# B&R Automation Studio project NAEUL004C00R13L518F00 (part 52)

#### Act_Main.st - Do Not Change!!!
```iecst
(** 2020-03-16 **)
ACTION Act_Main:

	IF bModuleNotOK = FALSE THEN
		CASE eStat OF

			LifterActIdle:
				IF eStatus <> Idle THEN	//Reset Data
					//Private
					fbStop(bEn := FALSE);
					fbRstAxisErr(bEn := FALSE);
					fbJog(bEn := FALSE);
					fbMovRel(bEn := FALSE);
					fbMovAbs(bEn := FALSE);
					fbHoming(bEn := FALSE);
					fbPwrOff(bEn := FALSE);
					fbPwrOn(bEn := FALSE);
					fbFullHm(bEn := FALSE);
					fbFullMovAbs(bEn := FALSE);
					fbFullMovRel(bEn := FALSE);
					fbSDOWrite(bEn := FALSE);
					fbTm(IN := FALSE);
					usiStep	:= 0;
					usiCount			:= 0;
					bNotInterruptible	:= FALSE;

					sStatTxt	:= a_sStatText[eStat];

				END_IF

				eStatus	:= Idle;

				IF EDGENEG(p_bManual) THEN
					fMotionCANRstCtrlWord(ADR(tyParamOutDriver));
				END_IF

			LifterActGoAPos:
				IF (eStatus = Idle OR eStatus = Busy) THEN

					eStatus	:= Busy;

					sStatTxt	:= a_sStatText[eStat];

					bNotInterruptible	:= TRUE;

					CASE usiStep OF
						0:	//Wait For Motion Parameter Update
							p_diMovePosInUM	:= p_diAPos;
							usiStep	:= 1;

						1:	//Check Position Difference
							IF tyParamOut.bPosDiff = TRUE THEN
								usiStep	:= 2;
							ELSE
								eStatus	:= Done;
							END_IF

						2:	//Move
							fbFullMovAbs.tyParamInDriver					:= tyParamInDriver;
							fbFullMovAbs.tyParamInMove.diPosInUM			:= p_diMovePosInUM;
							fbFullMovAbs.tyParamInMove.diDistInUM			:= p_diMoveDistInUM;
							fbFullMovAbs.tyParamInMove.diVelInUMPS			:= p_diMoveVelInUMPS;
							fbFullMovAbs.tyParamInMove.diAcc				:= p_diMoveAcc;
							fbFullMovAbs.tyParamInMove.diDec				:= p_diMoveDec;
							fbFullMovAbs.tyParamOut							:= tyParamOut;
							fbFullMovAbs(bEn := TRUE);

							IF fbFullMovAbs.udiStatus = 0 THEN
								eStatus	:= Done;
							ELSIF fbFullMovAbs.udiStatus < 65534 THEN
								eStatus		:= Error;

								IF fbFullMovAbs.udiStatus = 1401 THEN
									udiStatus	:= 10002;	//Power On Time Out While Going A Position
								ELSIF fbFullMovAbs.udiStatus = 1402 THEN
									udiStatus	:= 10003;	//Homing Time Out While Going A Position
								ELSIF fbFullMovAbs.udiStatus = 1403 THEN
									udiStatus	:= 10004;	//Move Absolute Time Out While Going A Position
								ELSIF fbFullMovAbs.udiStatus = 1405 THEN
									udiStatus	:= 10005;	//Stop Motion Time Out While Going A Position
								ELSIF fbFullMovAbs.udiStatus = 1408 THEN
									udiStatus	:= 10006;	//Axis Error Reset Failed While Going A Position
								ELSIF fbFullMovAbs.udiStatus = 1409 THEN
									udiStatus	:= 10007;	//Axis Error Occur In Move Absolute While Going A Position
								ELSIF fbFullMovAbs.udiStatus = 1411 THEN
									udiStatus	:= 10008;	//Axis Error Occur In Homing While Going A Position
								ELSIF fbFullMovAbs.udiStatus = 1412 THEN
									udiStatus	:= 10009;	//Homing Done But Home Flag Is Not Activated While Going A Position
								ELSIF fbFullMovAbs.udiStatus = 1413 THEN
									udiStatus	:= 10010;	//Forward Limit Activated In Homing While Going A Position
								ELSIF fbFullMovAbs.udiStatus = 1414 THEN
									udiStatus	:= 10011;	//Reverse Limit Activated In Homing While Going A Position
								ELSIF fbFullMovAbs.udiStatus = 1415 THEN
									udiStatus	:= 10012;	//Forward Limit Activated In Move Absolute While Going A Position
								ELSIF fbFullMovAbs.udiStatus = 1416 THEN
									udiStatus	:= 10013;	//Reverse Limit Activated In Move Absolute While Going A Position
								ELSE
									udiStatus	:= fbFullMovAbs.udiStatus;
								END_IF
							END_IF

					END_CASE

				END_IF

			LifterActGoBPos:
				IF (eStatus = Idle OR eStatus = Busy) THEN

					eStatus	:= Busy;

					sStatTxt	:= a_sStatText[eStat];

					bNotInterruptible	:= TRUE;

					CASE usiStep OF
						0:	//Wait For Motion Parameter Update
							p_diMovePosInUM	:= p_diBPos;
							usiStep	:= 1;

						1:	//Check Position Difference
							IF tyParamOut.bPosDiff = TRUE THEN
								usiStep	:= 2;
							ELSE
								eStatus	:= Done;
							END_IF

						2:	//Move
							fbFullMovAbs.tyParamInDriver					:= tyParamInDriver;
							fbFullMovAbs.tyParamInMove.diPosInUM			:= p_diMovePosInUM;
							fbFullMovAbs.tyParamInMove.diDistInUM			:= p_diMoveDistInUM;
							fbFullMovAbs.tyParamInMove.diVelInUMPS			:= p_diMoveVelInUMPS;
							fbFullMovAbs.tyParamInMove.diAcc				:= p_diMoveAcc;
							fbFullMovAbs.tyParamInMove.diDec				:= p_diMoveDec;
							fbFullMovAbs.tyParamOut							:= tyParamOut;
							fbFullMovAbs(bEn := TRUE);

							IF fbFullMovAbs.udiStatus = 0 THEN
								eStatus	:= Done;
							ELSIF fbFullMovAbs.udiStatus < 65534 THEN
								eStatus		:= Error;

								IF fbFullMovAbs.udiStatus = 1401 THEN
									udiStatus	:= 10029;	//Power On Time Out While Going B Position
								ELSIF fbFullMovAbs.udiStatus = 1402 THEN
									udiStatus	:= 10030;	//Homing Time Out While Going B Position
								ELSIF fbFullMovAbs.udiStatus = 1403 THEN
									udiStatus	:= 10031;	//Move Absolute Time Out While Going B Position
								ELSIF fbFullMovAbs.udiStatus = 1405 THEN
									udiStatus	:= 10032;	//Stop Motion Time Out While Going B Position
								ELSIF fbFullMovAbs.udiStatus = 1408 THEN
									udiStatus	:= 10033;	//Axis Error Reset Failed While Going B Position
								ELSIF fbFullMovAbs.udiStatus = 1409 THEN
									udiStatus	:= 10034;	//Axis Error Occur In Move Absolute While Going B Position
								ELSIF fbFullMovAbs.udiStatus = 1411 THEN
									udiStatus	:= 10035;	//Axis Error Occur In Homing While Going B Position
								ELSIF fbFullMovAbs.udiStatus = 1412 THEN
									udiStatus	:= 10036;	//Homing Done But Home Flag Is Not Activated While Going B Position
								ELSIF fbFullMovAbs.udiStatus = 1413 THEN
									udiStatus	:= 10037;	//Forward Limit Activated In Homing While Going B Position
								ELSIF fbFullMovAbs.udiStatus = 1414 THEN
									udiStatus	:= 10038;	//Reverse Limit Activated In Homing While Going B Position
								ELSIF fbFullMovAbs.udiStatus = 1415 THEN
									udiStatus	:= 10039;	//Forward Limit Activated In Move Absolute While Going B Position
								ELSIF fbFullMovAbs.udiStatus = 1416 THEN
									udiStatus	:= 10040;	//Reverse Limit Activated In Move Absolute While Going B Position
								ELSE
									udiStatus	:= fbFullMovAbs.udiStatus;
								END_IF
							END_IF

					END_CASE

				END_IF

			LifterActGoCPos:
				IF (eStatus = Idle OR eStatus = Busy) THEN

					eStatus	:= Busy;

					sStatTxt	:= a_sStatText[eStat];

					bNotInterruptible	:= TRUE;

					CASE usiStep OF
						0:	//Wait For Motion Parameter Update
							p_diMovePosInUM	:= p_diCPos;
							usiStep	:= 1;

						1:	//Check Position Difference
							IF tyParamOut.bPosDiff = TRUE THEN
								usiStep	:= 2;
							ELSE
								eStatus	:= Done;
							END_IF

						2:	//Move
							fbFullMovAbs.tyParamInDriver					:= tyParamInDriver;
							fbFullMovAbs.tyParamInMove.diPosInUM			:= p_diMovePosInUM;
							fbFullMovAbs.tyParamInMove.diDistInUM			:= p_diMoveDistInUM;
							fbFullMovAbs.tyParamInMove.diVelInUMPS			:= p_diMoveVelInUMPS;
							fbFullMovAbs.tyParamInMove.diAcc				:= p_diMoveAcc;
							fbFullMovAbs.tyParamInMove.diDec				:= p_diMoveDec;
							fbFullMovAbs.tyParamOut							:= tyParamOut;
							fbFullMovAbs(bEn := TRUE);

							IF fbFullMovAbs.udiStatus = 0 THEN
								eStatus	:= Done;
							ELSIF fbFullMovAbs.udiStatus < 65534 THEN
								eStatus		:= Error;

								IF fbFullMovAbs.udiStatus = 1401 THEN
									udiStatus	:= 10078;	//Power On Time Out While Going C Position
								ELSIF fbFullMovAbs.udiStatus = 1402 THEN
									udiStatus	:= 10079;	//Homing Time Out While Going C Position
								ELSIF fbFullMovAbs.udiStatus = 1403 THEN
									udiStatus	:= 10080;	//Move Absolute Time Out While Going C Position
								ELSIF fbFullMovAbs.udiStatus = 1405 THEN
									udiStatus	:= 10081;	//Stop Motion Time Out While Going C Position
								ELSIF fbFullMovAbs.udiStatus = 1408 THEN
									udiStatus	:= 10082;	//Axis Error Reset Failed While Going C Position
								ELSIF fbFullMovAbs.udiStatus = 1409 THEN
									udiStatus	:= 10083;	//Axis Error Occur In Move Absolute While Going C Position
								ELSIF fbFullMovAbs.udiStatus = 1411 THEN
									udiStatus	:= 10084;	//Axis Error Occur In Homing While Going C Position
								ELSIF fbFullMovAbs.udiStatus = 1412 THEN
									udiStatus	:= 10085;	//Homing Done But Home Flag Is Not Activated While Going C Position
								ELSIF fbFullMovAbs.udiStatus = 1413 THEN
									udiStatus	:= 10086;	//Forward Limit Activated In Homing While Going C Position
								ELSIF fbFullMovAbs.udiStatus = 1414 THEN
									udiStatus	:= 10087;	//Reverse Limit Activated In Homing While Going C Position
								ELSIF fbFullMovAbs.udiStatus = 1415 THEN
									udiStatus	:= 10088;	//Forward Limit Activated In Move Absolute While Going C Position
								ELSIF fbFullMovAbs.udiStatus = 1416 THEN
									udiStatus	:= 10089;	//Reverse Limit Activated In Move Absolute While Going C Position
								ELSE
									udiStatus	:= fbFullMovAbs.udiStatus;
								END_IF
							END_IF

					END_CASE

				END_IF

			LifterActGoDPos:
				IF (eStatus = Idle OR eStatus = Busy) THEN

					eStatus	:= Busy;

					sStatTxt	:= a_sStatText[eStat];

					bNotInterruptible	:= TRUE;

					CASE usiStep OF
						0:	//Wait For Motion Parameter Update
							p_diMovePosInUM	:= p_diDPos;
							usiStep	:= 1;

						1:	//Check Position Difference
							IF tyParamOut.bPosDiff = TRUE THEN
								usiStep	:= 2;
							ELSE
								eStatus	:= Done;
							END_IF

						2:	//Move
							fbFullMovAbs.tyParamInDriver					:= tyParamInDriver;
							fbFullMovAbs.tyParamInMove.diPosInUM			:= p_diMovePosInUM;
							fbFullMovAbs.tyParamInMove.diDistInUM			:= p_diMoveDistInUM;
							fbFullMovAbs.tyParamInMove.diVelInUMPS			:= p_diMoveVelInUMPS;
							fbFullMovAbs.tyParamInMove.diAcc				:= p_diMoveAcc;
							fbFullMovAbs.tyParamInMove.diDec				:= p_diMoveDec;
							fbFullMovAbs.tyParamOut							:= tyParamOut;
							fbFullMovAbs(bEn := TRUE);

							IF fbFullMovAbs.udiStatus = 0 THEN
								eStatus	:= Done;
							ELSIF fbFullMovAbs.udiStatus < 65534 THEN
								eStatus		:= Error;

								IF fbFullMovAbs.udiStatus = 1401 THEN
									udiStatus	:= 10090;	//Power On Time Out While Going D Position
								ELSIF fbFullMovAbs.udiStatus = 1402 THEN
									udiStatus	:= 10091;	//Homing Time Out While Going D Position
								ELSIF fbFullMovAbs.udiStatus = 1403 THEN
									udiStatus	:= 10092;	//Move Absolute Time Out While Going D Position
								ELSIF fbFullMovAbs.udiStatus = 1405 THEN
									udiStatus	:= 10093;	//Stop Motion Time Out While Going D Position
								ELSIF fbFullMovAbs.udiStatus = 1408 THEN
									udiStatus	:= 10094;	//Axis Error Reset Failed While Going D Position
								ELSIF fbFullMovAbs.udiStatus = 1409 THEN
									udiStatus	:= 10095;	//Axis Error Occur In Move Absolute While Going D Position
								ELSIF fbFullMovAbs.udiStatus = 1411 THEN
									udiStatus	:= 10096;	//Axis Error Occur In Homing While Going D Position
								ELSIF fbFullMovAbs.udiStatus = 1412 THEN
									udiStatus	:= 10097;	//Homing Done But Home Flag Is Not Activated While Going D Position
								ELSIF fbFullMovAbs.udiStatus = 1413 THEN
									udiStatus	:= 10098;	//Forward Limit Activated In Homing While Going D Position
								ELSIF fbFullMovAbs.udiStatus = 1414 THEN
									udiStatus	:= 10099;	//Reverse Limit Activated In Homing While Going D Position
								ELSIF fbFullMovAbs.udiStatus = 1415 THEN
									udiStatus	:= 10100;	//Forward Limit Activated In Move Absolute While Going D Position
								ELSIF fbFullMovAbs.udiStatus = 1416 THEN
									udiStatus	:= 10101;	//Reverse Limit Activated In Move Absolute While Going D Position
								ELSE
									udiStatus	:= fbFullMovAbs.udiStatus;
								END_IF
							END_IF

					END_CASE

				END_IF

			LifterActGoEPos:
				IF (eStatus = Idle OR eStatus = Busy) THEN

					eStatus	:= Busy;

					sStatTxt	:= a_sStatText[eStat];

					bNotInterruptible	:= TRUE;

					CASE usiStep OF
						0:	//Wait For Motion Parameter Update
							p_diMovePosInUM	:= p_diEPos;
							usiStep	:= 1;

						1:	//Check Position Difference
							IF tyParamOut.bPosDiff = TRUE THEN
								usiStep	:= 2;
							ELSE
								eStatus	:= Done;
							END_IF

						2:	//Move
							fbFullMovAbs.tyParamInDriver					:= tyParamInDriver;
							fbFullMovAbs.tyParamInMove.diPosInUM			:= p_diMovePosInUM;
							fbFullMovAbs.tyParamInMove.diDistInUM			:= p_diMoveDistInUM;
							fbFullMovAbs.tyParamInMove.diVelInUMPS			:= p_diMoveVelInUMPS;
							fbFullMovAbs.tyParamInMove.diAcc				:= p_diMoveAcc;
							fbFullMovAbs.tyParamInMove.diDec				:= p_diMoveDec;
							fbFullMovAbs.tyParamOut							:= tyParamOut;
							fbFullMovAbs(bEn := TRUE);

							IF fbFullMovAbs.udiStatus = 0 THEN
								eStatus	:= Done;
							ELSIF fbFullMovAbs.udiStatus < 65534 THEN
								eStatus		:= Error;

								IF fbFullMovAbs.udiStatus = 1401 THEN
									udiStatus	:= 10102;	//Power On Time Out While Going E Position
								ELSIF fbFullMovAbs.udiStatus = 1402 THEN
									udiStatus	:= 10103;	//Homing Time Out While Going E Position
								ELSIF fbFullMovAbs.udiStatus = 1403 THEN
									udiStatus	:= 10104;	//Move Absolute Time Out While Going E Position
								ELSIF fbFullMovAbs.udiStatus = 1405 THEN
									udiStatus	:= 10105;	//Stop Motion Time Out While Going E Position
								ELSIF fbFullMovAbs.udiStatus = 1408 THEN
									udiStatus	:= 10106;	//Axis Error Reset Failed While Going E Position
								ELSIF fbFullMovAbs.udiStatus = 1409 THEN
									udiStatus	:= 10107;	//Axis Error Occur In Move Absolute While Going E Position
								ELSIF fbFullMovAbs.udiStatus = 1411 THEN
									udiStatus	:= 10108;	//Axis Error Occur In Homing While Going E Position
								ELSIF fbFullMovAbs.udiStatus = 1412 THEN
									udiStatus	:= 10109;	//Homing Done But Home Flag Is Not Activated While Going E Position
								ELSIF fbFullMovAbs.udiStatus = 1413 THEN
									udiStatus	:= 10110;	//Forward Limit Activated In Homing While Going E Position
								ELSIF fbFullMovAbs.udiStatus = 1414 THEN
									udiStatus	:= 10111;	//Reverse Limit Activated In Homing While Going E Position
								ELSIF fbFullMovAbs.udiStatus = 1415 THEN
									udiStatus	:= 10112;	//Forward Limit Activated In Move Absolute While Going E Position
								ELSIF fbFullMovAbs.udiStatus = 1416 THEN
									udiStatus	:= 10113;	//Reverse Limit Activated In Move Absolute While Going E Position
								ELSE
									udiStatus	:= fbFullMovAbs.udiStatus;
								END_IF
							END_IF

					END_CASE

				END_IF

			LifterActGoFPos:
				IF (eStatus = Idle OR eStatus = Busy) THEN

					eStatus	:= Busy;

					sStatTxt	:= a_sStatText[eStat];

					bNotInterruptible	:= TRUE;

					CASE usiStep OF
						0:	//Wait For Motion Parameter Update
							p_diMovePosInUM	:= p_diFPos;
							usiStep	:= 1;

						1:	//Check Position Difference
							IF tyParamOut.bPosDiff = TRUE THEN
								usiStep	:= 2;
							ELSE
								eStatus	:= Done;
							END_IF

						2:	//Move
							fbFullMovAbs.tyParamInDriver					:= tyParamInDriver;
							fbFullMovAbs.tyParamInMove.diPosInUM			:= p_diMovePosInUM;
							fbFullMovAbs.tyParamInMove.diDistInUM			:= p_diMoveDistInUM;
							fbFullMovAbs.tyParamInMove.diVelInUMPS			:= p_diMoveVelInUMPS;
							fbFullMovAbs.tyParamInMove.diAcc				:= p_diMoveAcc;
							fbFullMovAbs.tyParamInMove.diDec				:= p_diMoveDec;
							fbFullMovAbs.tyParamOut							:= tyParamOut;
							fbFullMovAbs(bEn := TRUE);

							IF fbFullMovAbs.udiStatus = 0 THEN
								eStatus	:= Done;
							ELSIF fbFullMovAbs.udiStatus < 65534 THEN
								eStatus		:= Error;

								IF fbFullMovAbs.udiStatus = 1401 THEN
									udiStatus	:= 10114;	//Power On Time Out While Going F Position
								ELSIF fbFullMovAbs.udiStatus = 1402 THEN
									udiStatus	:= 10115;	//Homing Time Out While Going F Position
								ELSIF fbFullMovAbs.udiStatus = 1403 THEN
									udiStatus	:= 10116;	//Move Absolute Time Out While Going F Position
								ELSIF fbFullMovAbs.udiStatus = 1405 THEN
									udiStatus	:= 10117;	//Stop Motion Time Out While Going F Position
								ELSIF fbFullMovAbs.udiStatus = 1408 THEN
									udiStatus	:= 10118;	//Axis Error Reset Failed While Going F Position
								ELSIF fbFullMovAbs.udiStatus = 1409 THEN
									udiStatus	:= 10119;	//Axis Error Occur In Move Absolute While Going F Position
								ELSIF fbFullMovAbs.udiStatus = 1411 THEN
									udiStatus	:= 10120;	//Axis Error Occur In Homing While Going F Position
								ELSIF fbFullMovAbs.udiStatus = 1412 THEN
									udiStatus	:= 10121;	//Homing Done But Home Flag Is Not Activated While Going F Position
								ELSIF fbFullMovAbs.udiStatus = 1413 THEN
									udiStatus	:= 10122;	//Forward Limit Activated In Homing While Going F Position
								ELSIF fbFullMovAbs.udiStatus = 1414 THEN
									udiStatus	:= 10123;	//Reverse Limit Activated In Homing While Going F Position
								ELSIF fbFullMovAbs.udiStatus = 1415 THEN
									udiStatus	:= 10124;	//Forward Limit Activated In Move Absolute While Going F Position
								ELSIF fbFullMovAbs.udiStatus = 1416 THEN
									udiStatus	:= 10125;	//Reverse Limit Activated In Move Absolute While Going F Position
								ELSE
									udiStatus	:= fbFullMovAbs.udiStatus;
								END_IF
							END_IF

					END_CASE

				END_IF

			LifterActGoGPos:
				IF (eStatus = Idle OR eStatus = Busy) THEN

					eStatus	:= Busy;

					sStatTxt	:= a_sStatText[eStat];

					bNotInterruptible	:= TRUE;

					CASE usiStep OF
						0:	//Wait For Motion Parameter Update
							p_diMovePosInUM	:= p_diGPos;
							usiStep	:= 1;

						1:	//Check Position Difference
							IF tyParamOut.bPosDiff = TRUE THEN
								usiStep	:= 2;
							ELSE
								eStatus	:= Done;
							END_IF

						2:	//Move
							fbFullMovAbs.tyParamInDriver					:= tyParamInDriver;
							fbFullMovAbs.tyParamInMove.diPosInUM			:= p_diMovePosInUM;
							fbFullMovAbs.tyParamInMove.diDistInUM			:= p_diMoveDistInUM;
							fbFullMovAbs.tyParamInMove.diVelInUMPS			:= p_diMoveVelInUMPS;
							fbFullMovAbs.tyParamInMove.diAcc				:= p_diMoveAcc;
							fbFullMovAbs.tyParamInMove.diDec				:= p_diMoveDec;
							fbFullMovAbs.tyParamOut							:= tyParamOut;
							fbFullMovAbs(bEn := TRUE);

							IF fbFullMovAbs.udiStatus = 0 THEN
								eStatus	:= Done;
							ELSIF fbFullMovAbs.udiStatus < 65534 THEN
								eStatus		:= Error;

								IF fbFullMovAbs.udiStatus = 1401 THEN
									udiStatus	:= 10126;	//Power On Time Out While Going G Position
								ELSIF fbFullMovAbs.udiStatus = 1402 THEN
									udiStatus	:= 10127;	//Homing Time Out While Going G Position
								ELSIF fbFullMovAbs.udiStatus = 1403 THEN
									udiStatus	:= 10128;	//Move Absolute Time Out While Going G Position
								ELSIF fbFullMovAbs.udiStatus = 1405 THEN
									udiStatus	:= 10129;	//Stop Motion Time Out While Going G Position
								ELSIF fbFullMovAbs.udiStatus = 1408 THEN
									udiStatus	:= 10130;	//Axis Error Reset Failed While Going G Position
								ELSIF fbFullMovAbs.udiStatus = 1409 THEN
									udiStatus	:= 10131;	//Axis Error Occur In Move Absolute While Going G Position
								ELSIF fbFullMovAbs.udiStatus = 1411 THEN
									udiStatus	:= 10132;	//Axis Error Occur In Homing While Going G Position
								ELSIF fbFullMovAbs.udiStatus = 1412 THEN
									udiStatus	:= 10133;	//Homing Done But Home Flag Is Not Activated While Going G Position
								ELSIF fbFullMovAbs.udiStatus = 1413 THEN
									udiStatus	:= 10134;	//Forward Limit Activated In Homing While Going G Position
								ELSIF fbFullMovAbs.udiStatus = 1414 THEN
									udiStatus	:= 10135;	//Reverse Limit Activated In Homing While Going G Position
								ELSIF fbFullMovAbs.udiStatus = 1415 THEN
									udiStatus	:= 10136;	//Forward Limit Activated In Move Absolute While Going G Position
								ELSIF fbFullMovAbs.udiStatus = 1416 THEN
									udiStatus	:= 10137;	//Reverse Limit Activated In Move Absolute While Going G Position
								ELSE
									udiStatus	:= fbFullMovAbs.udiStatus;
								END_IF
							END_IF

					END_CASE

				END_IF

			LifterActGoHPos:
				IF (eStatus = Idle OR eStatus = Busy) THEN

					eStatus	:= Busy;

					sStatTxt	:= a_sStatText[eStat];

					bNotInterruptible	:= TRUE;

					CASE usiStep OF
						0:	//Wait For Motion Parameter Update
							p_diMovePosInUM	:= p_diHPos;
							usiStep	:= 1;

						1:	//Check Position Difference
							IF tyParamOut.bPosDiff = TRUE THEN
								usiStep	:= 2;
							ELSE
								eStatus	:= Done;
							END_IF

						2:	//Move
							fbFullMovAbs.tyParamInDriver					:= tyParamInDriver;
							fbFullMovAbs.tyParamInMove.diPosInUM			:= p_diMovePosInUM;
							fbFullMovAbs.tyParamInMove.diDistInUM			:= p_diMoveDistInUM;
							fbFullMovAbs.tyParamInMove.diVelInUMPS			:= p_diMoveVelInUMPS;
							fbFullMovAbs.tyParamInMove.diAcc				:= p_diMoveAcc;
							fbFullMovAbs.tyParamInMove.diDec				:= p_diMoveDec;
							fbFullMovAbs.tyParamOut							:= tyParamOut;
							fbFullMovAbs(bEn := TRUE);

							IF fbFullMovAbs.udiStatus = 0 THEN
								eStatus	:= Done;
							ELSIF fbFullMovAbs.udiStatus < 65534 THEN
								eStatus		:= Error;

								IF fbFullMovAbs.udiStatus = 1401 THEN
									udiStatus	:= 10138;	//Power On Time Out While Going H Position
								ELSIF fbFullMovAbs.udiStatus = 1402 THEN
									udiStatus	:= 10139;	//Homing Time Out While Going H Position
								ELSIF fbFullMovAbs.udiStatus = 1403 THEN
									udiStatus	:= 10140;	//Move Absolute Time Out While Going H Position
								ELSIF fbFullMovAbs.udiStatus = 1405 THEN
									udiStatus	:= 10141;	//Stop Motion Time Out While Going H Position
								ELSIF fbFullMovAbs.udiStatus = 1408 THEN
									udiStatus	:= 10142;	//Axis Error Reset Failed While Going H Position
								ELSIF fbFullMovAbs.udiStatus = 1409 THEN
									udiStatus	:= 10143;	//Axis Error Occur In Move Absolute While Going H Position
								ELSIF fbFullMovAbs.udiStatus = 1411 THEN
									udiStatus	:= 10144;	//Axis Error Occur In Homing While Going H Position
								ELSIF fbFullMovAbs.udiStatus = 1412 THEN
									udiStatus	:= 10145;	//Homing Done But Home Flag Is Not Activated While Going H Position
								ELSIF fbFullMovAbs.udiStatus = 1413 THEN
									udiStatus	:= 10146;	//Forward Limit Activated In Homing While Going H Position
								ELSIF fbFullMovAbs.udiStatus = 1414 THEN
									udiStatus	:= 10147;	//Reverse Limit Activated In Homing While Going H Position
								ELSIF fbFullMovAbs.udiStatus = 1415 THEN
									udiStatus	:= 10148;	//Forward Limit Activated In Move Absolute While Going H Position
								ELSIF fbFullMovAbs.udiStatus = 1416 THEN
									udiStatus	:= 10149;	//Reverse Limit Activated In Move Absolute While Going H Position
								ELSE
									udiStatus	:= fbFullMovAbs.udiStatus;
								END_IF
							END_IF

					END_CASE

				END_IF

			LifterActGoASltPos:
				IF (eStatus = Idle OR eStatus = Busy) THEN

					eStatus	:= Busy;

					sStatTxt	:= a_sStatText[eStat];

					bNotInterruptible	:= TRUE;

					CASE usiStep OF
						0:	//Wait For Motion Parameter Update
							p_diMovePosInUM	:= fLifterSltToPosInUMBtmMin(p_diGoASlt , p_diASltToSltDist , p_diASlt1Pos);
							usiStep	:= 1;

						1:	//Check Position Difference
							IF tyParamOut.bPosDiff = TRUE THEN
								usiStep	:= 2;
							ELSE
								eStatus	:= Done;
							END_IF

						2:	//Move
							fbFullMovAbs.tyParamInDriver					:= tyParamInDriver;
							fbFullMovAbs.tyParamInMove.diPosInUM			:= p_diMovePosInUM;
							fbFullMovAbs.tyParamInMove.diDistInUM			:= p_diMoveDistInUM;
							fbFullMovAbs.tyParamInMove.diVelInUMPS			:= p_diMoveVelInUMPS;
							fbFullMovAbs.tyParamInMove.diAcc				:= p_diMoveAcc;
							fbFullMovAbs.tyParamInMove.diDec				:= p_diMoveDec;
							fbFullMovAbs.tyParamOut							:= tyParamOut;
							fbFullMovAbs(bEn := TRUE);

							IF fbFullMovAbs.udiStatus = 0 THEN
								eStatus	:= Done;
							ELSIF fbFullMovAbs.udiStatus < 65534 THEN
								eStatus		:= Error;

								IF fbFullMovAbs.udiStatus = 1401 THEN
									udiStatus	:= 10041;	//Power On Time Out While Going New A Slot Position
								ELSIF fbFullMovAbs.udiStatus = 1402 THEN
									udiStatus	:= 10042;	//Homing Time Out While Going New A Slot Position
								ELSIF fbFullMovAbs.udiStatus = 1403 THEN
									udiStatus	:= 10043;	//Move Absolute Time Out While Going New A Slot Position
								ELSIF fbFullMovAbs.udiStatus = 1405 THEN
									udiStatus	:= 10044;	//Stop Motion Time Out While Going New A Slot Position
								ELSIF fbFullMovAbs.udiStatus = 1408 THEN
									udiStatus	:= 10045;	//Axis Error Reset Failed While Going New A Slot Position
								ELSIF fbFullMovAbs.udiStatus = 1409 THEN
									udiStatus	:= 10046;	//Axis Error Occur In Move Absolute While Going New A Slot Position
								ELSIF fbFullMovAbs.udiStatus = 1411 THEN
									udiStatus	:= 10047;	//Axis Error Occur In Homing While Going New A Slot Position
								ELSIF fbFullMovAbs.udiStatus = 1412 THEN
									udiStatus	:= 10048;	//Homing Done But Home Flag Is Not Activated While Going New A Slot Position
								ELSIF fbFullMovAbs.udiStatus = 1413 THEN
									udiStatus	:= 10049;	//Forward Limit Activated In Homing While Going New A Slot Position
								ELSIF fbFullMovAbs.udiStatus = 1414 THEN
									udiStatus	:= 10050;	//Reverse Limit Activated In Homing While Going New A Slot Position
								ELSIF fbFullMovAbs.udiStatus = 1415 THEN
									udiStatus	:= 10051;	//Forward Limit Activated In Move Absolute While Going New A Slot Position
								ELSIF fbFullMovAbs.udiStatus = 1416 THEN
									udiStatus	:= 10052;	//Reverse Limit Activated In Move Absolute While Going New A Slot Position
								ELSE
									udiStatus	:= fbFullMovAbs.udiStatus;
								END_IF
							END_IF

					END_CASE

				END_IF

			LifterActGoNxtASltPos:
				IF (eStatus = Idle OR eStatus = Busy) THEN

					eStatus	:= Busy;

					sStatTxt	:= a_sStatText[eStat];

					bNotInterruptible	:= TRUE;

					CASE usiStep OF
						0:	//Wait For Motion Parameter Update
							diExpectSlt		:= fLifterPosInUMToSltBtmMin(tyParamOut.diActualPosInUM , p_diASltToSltDist , p_diASlt1Pos);
							diExpectPosInUM	:= fLifterSltToPosInUMBtmMin(diExpectSlt , p_diASltToSltDist , p_diASlt1Pos);

							IF ABS(tyParamOut.diActualPosInUM - diExpectPosInUM) < 50 THEN
								p_diGoASlt		:= diExpectSlt + 1;
								p_diMovePosInUM	:= fLifterSltToPosInUMBtmMin(p_diGoASlt , p_diASltToSltDist , p_diASlt1Pos);

							ELSIF tyParamOut.diActualPosInUM > diExpectPosInUM THEN
								p_diGoASlt		:= diExpectSlt;
								p_diMovePosInUM	:= fLifterSltToPosInUMBtmMin(p_diGoASlt , p_diASltToSltDist , p_diASlt1Pos);

							ELSIF tyParamOut.diActualPosInUM < diExpectPosInUM THEN
								p_diGoASlt		:= diExpectSlt + 1;
								p_diMovePosInUM	:= fLifterSltToPosInUMBtmMin(p_diGoASlt , p_diASltToSltDist , p_diASlt1Pos);

							END_IF

							usiStep	:= 1;

						1:	//Check Position Difference
							IF tyParamOut.bPosDiff = TRUE THEN
								usiStep	:= 2;
							ELSE
								eStatus	:= Done;
							END_IF

						2:	//Move
							fbFullMovAbs.tyParamInDriver					:= tyParamInDriver;
							fbFullMovAbs.tyParamInMove.diPosInUM			:= p_diMovePosInUM;
							fbFullMovAbs.tyParamInMove.diDistInUM			:= p_diMoveDistInUM;
							fbFullMovAbs.tyParamInMove.diVelInUMPS			:= p_diMoveVelInUMPS;
							fbFullMovAbs.tyParamInMove.diAcc				:= p_diMoveAcc;
							fbFullMovAbs.tyParamInMove.diDec				:= p_diMoveDec;
							fbFullMovAbs.tyParamOut							:= tyParamOut;
							fbFullMovAbs(bEn := TRUE);

							IF fbFullMovAbs.udiStatus = 0 THEN
								eStatus	:= Done;
							ELSIF fbFullMovAbs.udiStatus < 65534 THEN
								eStatus		:= Error;

								IF fbFullMovAbs.udiStatus = 1401 THEN
									udiStatus	:= 10053;	//Power On Time Out While Going Next A Slot Position
								ELSIF fbFullMovAbs.udiStatus = 1402 THEN
									udiStatus	:= 10054;	//Homing Time Out While Going Next A Slot Position
								ELSIF fbFullMovAbs.udiStatus = 1403 THEN
									udiStatus	:= 10055;	//Move Absolute Time Out While Going Next A Slot Position
								ELSIF fbFullMovAbs.udiStatus = 1405 THEN
									udiStatus	:= 10056;	//Stop Motion Time Out While Going Next A Slot Position
								ELSIF fbFullMovAbs.udiStatus = 1408 THEN
									udiStatus	:= 10057;	//Axis Error Reset Failed While Going Next A Slot Position
								ELSIF fbFullMovAbs.udiStatus = 1409 THEN
									udiStatus	:= 10058;	//Axis Error Occur In Move Absolute While Going Next A Slot Position
								ELSIF fbFullMovAbs.udiStatus = 1411 THEN
									udiStatus	:= 10059;	//Axis Error Occur In Homing While Going Next A Slot Position
								ELSIF fbFullMovAbs.udiStatus = 1412 THEN
									udiStatus	:= 10060;	//Homing Done But Home Flag Is Not Activated While Going Next A Slot Position
								ELSIF fbFullMovAbs.udiStatus = 1413 THEN
									udiStatus	:= 10061;	//Forward Limit Activated In Homing While Going Next A Slot Position
								ELSIF fbFullMovAbs.udiStatus = 1414 THEN
									udiStatus	:= 10062;	//Reverse Limit Activated In Homing While Going Next A Slot Position
								ELSIF fbFullMovAbs.udiStatus = 1415 THEN
									udiStatus	:= 10063;	//Forward Limit Activated In Move Absolute While Going Next A Slot Position
								ELSIF fbFullMovAbs.udiStatus = 1416 THEN
									udiStatus	:= 10064;	//Reverse Limit Activated In Move Absolute While Going Next A Slot Position
								ELSE
									udiStatus	:= fbFullMovAbs.udiStatus;
								END_IF
							END_IF

					END_CASE

				END_IF

			LifterActGoPrevASltPos:
				IF (eStatus = Idle OR eStatus = Busy) THEN

					eStatus	:= Busy;

					sStatTxt	:= a_sStatText[eStat];

					bNotInterruptible	:= TRUE;

					CASE usiStep OF
						0:	//Wait For Motion Parameter Update
							diExpectSlt		:= fLifterPosInUMToSltBtmMin(tyParamOut.diActualPosInUM , p_diASltToSltDist , p_diASlt1Pos);
							diExpectPosInUM	:= fLifterSltToPosInUMBtmMin(diExpectSlt , p_diASltToSltDist , p_diASlt1Pos);

							IF ABS(tyParamOut.diActualPosInUM - diExpectPosInUM) < 50 THEN
								p_diGoASlt		:= diExpectSlt - 1;
								p_diMovePosInUM	:= fLifterSltToPosInUMBtmMin(p_diGoASlt , p_diASltToSltDist , p_diASlt1Pos);

							ELSIF tyParamOut.diActualPosInUM > diExpectPosInUM THEN
								p_diGoASlt		:= diExpectSlt - 1;
								p_diMovePosInUM	:= fLifterSltToPosInUMBtmMin(p_diGoASlt , p_diASltToSltDist , p_diASlt1Pos);

							ELSIF tyParamOut.diActualPosInUM < diExpectPosInUM THEN
								p_diGoASlt		:= diExpectSlt;
								p_diMovePosInUM	:= fLifterSltToPosInUMBtmMin(p_diGoASlt , p_diASltToSltDist , p_diASlt1Pos);

							END_IF

							usiStep	:= 1;

						1:	//Check Position Difference
							IF tyParamOut.bPosDiff = TRUE THEN
								usiStep	:= 2;
							ELSE
								eStatus	:= Done;
							END_IF

						2:	//Move
							fbFullMovAbs.tyParamInDriver					:= tyParamInDriver;
							fbFullMovAbs.tyParamInMove.diPosInUM			:= p_diMovePosInUM;
							fbFullMovAbs.tyParamInMove.diDistInUM			:= p_diMoveDistInUM;
							fbFullMovAbs.tyParamInMove.diVelInUMPS			:= p_diMoveVelInUMPS;
							fbFullMovAbs.tyParamInMove.diAcc				:= p_diMoveAcc;
							fbFullMovAbs.tyParamInMove.diDec				:= p_diMoveDec;
							fbFullMovAbs.tyParamOut							:= tyParamOut;
							fbFullMovAbs(bEn := TRUE);

							IF fbFullMovAbs.udiStatus = 0 THEN
								eStatus	:= Done;
							ELSIF fbFullMovAbs.udiStatus < 65534 THEN
								eStatus		:= Error;

								IF fbFullMovAbs.udiStatus = 1401 THEN
									udiStatus	:= 10065;	//Power On Time Out While Going Previous A Slot Position
								ELSIF fbFullMovAbs.udiStatus = 1402 THEN
									udiStatus	:= 10066;	//Homing Time Out While Going Previous A Slot Position
								ELSIF fbFullMovAbs.udiStatus = 1403 THEN
									udiStatus	:= 10067;	//Move Absolute Time Out While Going Previous A Slot Position
								ELSIF fbFullMovAbs.udiStatus = 1405 THEN
									udiStatus	:= 10068;	//Stop Motion Time Out While Going Previous A Slot Position
								ELSIF fbFullMovAbs.udiStatus = 1408 THEN
									udiStatus	:= 10069;	//Axis Error Reset Failed While Going Previous A Slot Position
								ELSIF fbFullMovAbs.udiStatus = 1409 THEN
									udiStatus	:= 10070;	//Axis Error Occur In Move Absolute While Going Previous A Slot Position
								ELSIF fbFullMovAbs.udiStatus = 1411 THEN
									udiStatus	:= 10071;	//Axis Error Occur In Homing While Going Previous A Slot Position
								ELSIF fbFullMovAbs.udiStatus = 1412 THEN
									udiStatus	:= 10072;	//Homing Done But Home Flag Is Not Activated While Going Previous A Slot Position
								ELSIF fbFullMovAbs.udiStatus = 1413 THEN
									udiStatus	:= 10073;	//Forward Limit Activated In Homing While Going Previous A Slot Position
								ELSIF fbFullMovAbs.udiStatus = 1414 THEN
									udiStatus	:= 10074;	//Reverse Limit Activated In Homing While Going Previous A Slot Position
								ELSIF fbFullMovAbs.udiStatus = 1415 THEN
									udiStatus	:= 10075;	//Forward Limit Activated In Move Absolute While Going Previous A Slot Position
								ELSIF fbFullMovAbs.udiStatus = 1416 THEN
									udiStatus	:= 10076;	//Reverse Limit Activated In Move Absolute While Going Previous A Slot Position
								ELSE
									udiStatus	:= fbFullMovAbs.udiStatus;
								END_IF
							END_IF

					END_CASE

				END_IF

			LifterActGoBSltPos:
				IF (eStatus = Idle OR eStatus = Busy) THEN

					eStatus	:= Busy;

					sStatTxt	:= a_sStatText[eStat];

					bNotInterruptible	:= TRUE;

					CASE usiStep OF
						0:	//Wait For Motion Parameter Update
							p_diMovePosInUM	:= fLifterSltToPosInUMBtmMin(p_diGoBSlt , p_diBSltToSltDist , p_diBSlt1Pos);
							usiStep	:= 1;

						1:	//Check Position Difference
							IF tyParamOut.bPosDiff = TRUE THEN
								usiStep	:= 2;
							ELSE
								eStatus	:= Done;
							END_IF

						2:	//Move
							fbFullMovAbs.tyParamInDriver					:= tyParamInDriver;
							fbFullMovAbs.tyParamInMove.diPosInUM			:= p_diMovePosInUM;
							fbFullMovAbs.tyParamInMove.diDistInUM			:= p_diMoveDistInUM;
							fbFullMovAbs.tyParamInMove.diVelInUMPS			:= p_diMoveVelInUMPS;
							fbFullMovAbs.tyParamInMove.diAcc				:= p_diMoveAcc;
							fbFullMovAbs.tyParamInMove.diDec				:= p_diMoveDec;
							fbFullMovAbs.tyParamOut							:= tyParamOut;
							fbFullMovAbs(bEn := TRUE);

							IF fbFullMovAbs.udiStatus = 0 THEN
								eStatus	:= Done;
							ELSIF fbFullMovAbs.udiStatus < 65534 THEN
								eStatus		:= Error;

								IF fbFullMovAbs.udiStatus = 1401 THEN
									udiStatus	:= 10150;	//Power On Time Out While Going New B Slot Position
								ELSIF fbFullMovAbs.udiStatus = 1402 THEN
									udiStatus	:= 10151;	//Homing Time Out While Going New B Slot Position
								ELSIF fbFullMovAbs.udiStatus = 1403 THEN
									udiStatus	:= 10152;	//Move Absolute Time Out While Going New B Slot Position
								ELSIF fbFullMovAbs.udiStatus = 1405 THEN
									udiStatus	:= 10153;	//Stop Motion Time Out While Going New B Slot Position
								ELSIF fbFullMovAbs.udiStatus = 1408 THEN
									udiStatus	:= 10154;	//Axis Error Reset Failed While Going New B Slot Position
								ELSIF fbFullMovAbs.udiStatus = 1409 THEN
									udiStatus	:= 10155;	//Axis Error Occur In Move Absolute While Going New B Slot Position
								ELSIF fbFullMovAbs.udiStatus = 1411 THEN
									udiStatus	:= 10156;	//Axis Error Occur In Homing While Going New B Slot Position
								ELSIF fbFullMovAbs.udiStatus = 1412 THEN
									udiStatus	:= 10157;	//Homing Done But Home Flag Is Not Activated While Going New B Slot Position
								ELSIF fbFullMovAbs.udiStatus = 1413 THEN
									udiStatus	:= 10158;	//Forward Limit Activated In Homing While Going New B Slot Position
								ELSIF fbFullMovAbs.udiStatus = 1414 THEN
									udiStatus	:= 10159;	//Reverse Limit Activated In Homing While Going New B Slot Position
								ELSIF fbFullMovAbs.udiStatus = 1415 THEN
									udiStatus	:= 10160;	//Forward Limit Activated In Move Absolute While Going New B Slot Position
								ELSIF fbFullMovAbs.udiStatus = 1416 THEN
									udiStatus	:= 10161;	//Reverse Limit Activated In Move Absolute While Going New B Slot Position
								ELSE
									udiStatus	:= fbFullMovAbs.udiStatus;
								END_IF
							END_IF

					END_CASE

				END_IF

			LifterActGoNxtBSltPos:
				IF (eStatus = Idle OR eStatus = Busy) THEN

					eStatus	:= Busy;

					sStatTxt	:= a_sStatText[eStat];

					bNotInterruptible	:= TRUE;

					CASE usiStep OF
						0:	//Wait For Motion Parameter Update
							diExpectSlt		:= fLifterPosInUMToSltBtmMin(tyParamOut.diActualPosInUM , p_diBSltToSltDist , p_diBSlt1Pos);
							diExpectPosInUM	:= fLifterSltToPosInUMBtmMin(diExpectSlt , p_diBSltToSltDist , p_diBSlt1Pos);

							IF ABS(tyParamOut.diActualPosInUM - diExpectPosInUM) < 50 THEN
								p_diGoBSlt		:= diExpectSlt + 1;
								p_diMovePosInUM	:= fLifterSltToPosInUMBtmMin(p_diGoBSlt , p_diBSltToSltDist , p_diBSlt1Pos);

							ELSIF tyParamOut.diActualPosInUM > diExpectPosInUM THEN
								p_diGoBSlt		:= diExpectSlt;
								p_diMovePosInUM	:= fLifterSltToPosInUMBtmMin(p_diGoBSlt , p_diBSltToSltDist , p_diBSlt1Pos);

							ELSIF tyParamOut.diActualPosInUM < diExpectPosInUM THEN
								p_diGoBSlt		:= diExpectSlt + 1;
								p_diMovePosInUM	:= fLifterSltToPosInUMBtmMin(p_diGoBSlt , p_diBSltToSltDist , p_diBSlt1Pos);

							END_IF

							usiStep	:= 1;

						1:	//Check Position Difference
							IF tyParamOut.bPosDiff = TRUE THEN
								usiStep	:= 2;
							ELSE
								eStatus	:= Done;
							END_IF

						2:	//Move
							fbFullMovAbs.tyParamInDriver					:= tyParamInDriver;
							fbFullMovAbs.tyParamInMove.diPosInUM			:= p_diMovePosInUM;
							fbFullMovAbs.tyParamInMove.diDistInUM			:= p_diMoveDistInUM;
							fbFullMovAbs.tyParamInMove.diVelInUMPS			:= p_diMoveVelInUMPS;
							fbFullMovAbs.tyParamInMove.diAcc				:= p_diMoveAcc;
							fbFullMovAbs.tyParamInMove.diDec				:= p_diMoveDec;
							fbFullMovAbs.tyParamOut							:= tyParamOut;
							fbFullMovAbs(bEn := TRUE);

							IF fbFullMovAbs.udiStatus = 0 THEN
								eStatus	:= Done;
							ELSIF fbFullMovAbs.udiStatus < 65534 THEN
								eStatus		:= Error;

								IF fbFullMovAbs.udiStatus = 1401 THEN
									udiStatus	:= 10162;	//Power On Time Out While Going Next B Slot Position
								ELSIF fbFullMovAbs.udiStatus = 1402 THEN
									udiStatus	:= 10163;	//Homing Time Out While Going Next B Slot Position
								ELSIF fbFullMovAbs.udiStatus = 1403 THEN
									udiStatus	:= 10164;	//Move Absolute Time Out While Going Next B Slot Position
								ELSIF fbFullMovAbs.udiStatus = 1405 THEN
									udiStatus	:= 10165;	//Stop Motion Time Out While Going Next B Slot Position
								ELSIF fbFullMovAbs.udiStatus = 1408 THEN
									udiStatus	:= 10166;	//Axis Error Reset Failed While Going Next B Slot Position
								ELSIF fbFullMovAbs.udiStatus = 1409 THEN
									udiStatus	:= 10167;	//Axis Error Occur In Move Absolute While Going Next B Slot Position
								ELSIF fbFullMovAbs.udiStatus = 1411 THEN
									udiStatus	:= 10168;	//Axis Error Occur In Homing While Going Next B Slot Position
								ELSIF fbFullMovAbs.udiStatus = 1412 THEN
									udiStatus	:= 10169;	//Homing Done But Home Flag Is Not Activated While Going Next B Slot Position
								ELSIF fbFullMovAbs.udiStatus = 1413 THEN
									udiStatus	:= 10170;	//Forward Limit Activated In Homing While Going Next B Slot Position
								ELSIF fbFullMovAbs.udiStatus = 1414 THEN
									udiStatus	:= 10171;	//Reverse Limit Activated In Homing While Going Next B Slot Position
								ELSIF fbFullMovAbs.udiStatus = 1415 THEN
									udiStatus	:= 10172;	//Forward Limit Activated In Move Absolute While Going Next B Slot Position
								ELSIF fbFullMovAbs.udiStatus = 1416 THEN
									udiStatus	:= 10173;	//Reverse Limit Activated In Move Absolute While Going Next B Slot Position
								ELSE
									udiStatus	:= fbFullMovAbs.udiStatus;
								END_IF
							END_IF

					END_CASE

				END_IF

			LifterActGoPrevBSltPos:
				IF (eStatus = Idle OR eStatus = Busy) THEN

					eStatus	:= Busy;

					sStatTxt	:= a_sStatText[eStat];

					bNotInterruptible	:= TRUE;

					CASE usiStep OF
						0:	//Wait For Motion Parameter Update
							diExpectSlt		:= fLifterPosInUMToSltBtmMin(tyParamOut.diActualPosInUM , p_diBSltToSltDist , p_diBSlt1Pos);
							diExpectPosInUM	:= fLifterSltToPosInUMBtmMin(diExpectSlt , p_diBSltToSltDist , p_diBSlt1Pos);

							IF ABS(tyParamOut.diActualPosInUM - diExpectPosInUM) < 50 THEN
								p_diGoBSlt		:= diExpectSlt - 1;
								p_diMovePosInUM	:= fLifterSltToPosInUMBtmMin(p_diGoBSlt , p_diBSltToSltDist , p_diBSlt1Pos);

							ELSIF tyParamOut.diActualPosInUM > diExpectPosInUM THEN
								p_diGoBSlt		:= diExpectSlt - 1;
								p_diMovePosInUM	:= fLifterSltToPosInUMBtmMin(p_diGoBSlt , p_diBSltToSltDist , p_diBSlt1Pos);

							ELSIF tyParamOut.diActualPosInUM < diExpectPosInUM THEN
								p_diGoBSlt		:= diExpectSlt;
								p_diMovePosInUM	:= fLifterSltToPosInUMBtmMin(p_diGoBSlt , p_diBSltToSltDist , p_diBSlt1Pos);

							END_IF

							usiStep	:= 1;

						1:	//Check Position Difference
							IF tyParamOut.bPosDiff = TRUE THEN
								usiStep	:= 2;
							ELSE
								eStatus	:= Done;
							END_IF

						2:	//Move
							fbFullMovAbs.tyParamInDriver					:= tyParamInDriver;
							fbFullMovAbs.tyParamInMove.diPosInUM			:= p_diMovePosInUM;
							fbFullMovAbs.tyParamInMove.diDistInUM			:= p_diMoveDistInUM;
							fbFullMovAbs.tyParamInMove.diVelInUMPS			:= p_diMoveVelInUMPS;
							fbFullMovAbs.tyParamInMove.diAcc				:= p_diMoveAcc;
							fbFullMovAbs.tyParamInMove.diDec				:= p_diMoveDec;
							fbFullMovAbs.tyParamOut							:= tyParamOut;
							fbFullMovAbs(bEn := TRUE);

							IF fbFullMovAbs.udiStatus = 0 THEN
								eStatus	:= Done;
							ELSIF fbFullMovAbs.udiStatus < 65534 THEN
								eStatus		:= Error;

								IF fbFullMovAbs.udiStatus = 1401 THEN
									udiStatus	:= 10174;	//Power On Time Out While Going Previous B Slot Position
								ELSIF fbFullMovAbs.udiStatus = 1402 THEN
									udiStatus	:= 10175;	//Homing Time Out While Going Previous B Slot Position
								ELSIF fbFullMovAbs.udiStatus = 1403 THEN
									udiStatus	:= 10176;	//Move Absolute Time Out While Going Previous B Slot Position
								ELSIF fbFullMovAbs.udiStatus = 1405 THEN
									udiStatus	:= 10177;	//Stop Motion Time Out While Going Previous B Slot Position
								ELSIF fbFullMovAbs.udiStatus = 1408 THEN
									udiStatus	:= 10178;	//Axis Error Reset Failed While Going Previous B Slot Position
								ELSIF fbFullMovAbs.udiStatus = 1409 THEN
									udiStatus	:= 10179;	//Axis Error Occur In Move Absolute While Going Previous B Slot Position
								ELSIF fbFullMovAbs.udiStatus = 1411 THEN
									udiStatus	:= 10180;	//Axis Error Occur In Homing While Going Previous B Slot Position
								ELSIF fbFullMovAbs.udiStatus = 1412 THEN
									udiStatus	:= 10181;	//Homing Done But Home Flag Is Not Activated While Going Previous B Slot Position
								ELSIF fbFullMovAbs.udiStatus = 1413 THEN
									udiStatus	:= 10182;	//Forward Limit Activated In Homing While Going Previous B Slot Position
								ELSIF fbFullMovAbs.udiStatus = 1414 THEN
									udiStatus	:= 10183;	//Reverse Limit Activated In Homing While Going Previous B Slot Position
								ELSIF fbFullMovAbs.udiStatus = 1415 THEN
									udiStatus	:= 10184;	//Forward Limit Activated In Move Absolute While Going Previous B Slot Position
								ELSIF fbFullMovAbs.udiStatus = 1416 THEN
									udiStatus	:= 10185;	//Reverse Limit Activated In Move Absolute While Going Previous B Slot Position
								ELSE
									udiStatus	:= fbFullMovAbs.udiStatus;
								END_IF
							END_IF

					END_CASE

				END_IF

			LifterActGoCSltPos:
				IF (eStatus = Idle OR eStatus = Busy) THEN

					eStatus	:= Busy;

					sStatTxt	:= a_sStatText[eStat];

					bNotInterruptible	:= TRUE;

					CASE usiStep OF
						0:	//Wait For Motion Parameter Update
							p_diMovePosInUM	:= fLifterSltToPosInUMBtmMin(p_diGoCSlt , p_diCSltToSltDist , p_diCSlt1Pos);
							usiStep	:= 1;

						1:	//Check Position Difference
							IF tyParamOut.bPosDiff = TRUE THEN
								usiStep	:= 2;
							ELSE
								eStatus	:= Done;
							END_IF

						2:	//Move
							fbFullMovAbs.tyParamInDriver					:= tyParamInDriver;
							fbFullMovAbs.tyParamInMove.diPosInUM			:= p_diMovePosInUM;
							fbFullMovAbs.tyParamInMove.diDistInUM			:= p_diMoveDistInUM;
							fbFullMovAbs.tyParamInMove.diVelInUMPS			:= p_diMoveVelInUMPS;
							fbFullMovAbs.tyParamInMove.diAcc				:= p_diMoveAcc;
							fbFullMovAbs.tyParamInMove.diDec				:= p_diMoveDec;
							fbFullMovAbs.tyParamOut							:= tyParamOut;
							fbFullMovAbs(bEn := TRUE);

							IF fbFullMovAbs.udiStatus = 0 THEN
								eStatus	:= Done;
							ELSIF fbFullMovAbs.udiStatus < 65534 THEN
								eStatus		:= Error;

								IF fbFullMovAbs.udiStatus = 1401 THEN
									udiStatus	:= 10186;	//Power On Time Out While Going New C Slot Position
								ELSIF fbFullMovAbs.udiStatus = 1402 THEN
									udiStatus	:= 10187;	//Homing Time Out While Going New C  Slot Position
								ELSIF fbFullMovAbs.udiStatus = 1403 THEN
									udiStatus	:= 10188;	//Move Absolute Time Out While Going New C  Slot Position
								ELSIF fbFullMovAbs.udiStatus = 1405 THEN
									udiStatus	:= 10189;	//Stop Motion Time Out While Going New C  Slot Position
								ELSIF fbFullMovAbs.udiStatus = 1408 THEN
									udiStatus	:= 10190;	//Axis Error Reset Failed While Going New C  Slot Position
								ELSIF fbFullMovAbs.udiStatus = 1409 THEN
									udiStatus	:= 10191;	//Axis Error Occur In Move Absolute While Going New C  Slot Position
								ELSIF fbFullMovAbs.udiStatus = 1411 THEN
									udiStatus	:= 10192;	//Axis Error Occur In Homing While Going New C  Slot Position
								ELSIF fbFullMovAbs.udiStatus = 1412 THEN
									udiStatus	:= 10193;	//Homing Done But Home Flag Is Not Activated While Going New C  Slot Position
								ELSIF fbFullMovAbs.udiStatus = 1413 THEN
									udiStatus	:= 10194;	//Forward Limit Activated In Homing While Going New C  Slot Position
								ELSIF fbFullMovAbs.udiStatus = 1414 THEN
									udiStatus	:= 10195;	//Reverse Limit Activated In Homing While Going New C  Slot Position
								ELSIF fbFullMovAbs.udiStatus = 1415 THEN
									udiStatus	:= 10196;	//Forward Limit Activated In Move Absolute While Going New C  Slot Position
								ELSIF fbFullMovAbs.udiStatus = 1416 THEN
									udiStatus	:= 10197;	//Reverse Limit Activated In Move Absolute While Going New C  Slot Position
								ELSE
									udiStatus	:= fbFullMovAbs.udiStatus;
								END_IF
							END_IF

					END_CASE

				END_IF

			LifterActGoNxtCSltPos:
				IF (eStatus = Idle OR eStatus = Busy) THEN

					eStatus	:= Busy;

					sStatTxt	:= a_sStatText[eStat];

					bNotInterruptible	:= TRUE;

					CASE usiStep OF
						0:	//Wait For Motion Parameter Update
							diExpectSlt		:= fLifterPosInUMToSltBtmMin(tyParamOut.diActualPosInUM , p_diCSltToSltDist , p_diCSlt1Pos);
							diExpectPosInUM	:= fLifterSltToPosInUMBtmMin(diExpectSlt , p_diCSltToSltDist , p_diCSlt1Pos);

							IF ABS(tyParamOut.diActualPosInUM - diExpectPosInUM) < 50 THEN
								p_diGoCSlt		:= diExpectSlt + 1;
								p_diMovePosInUM	:= fLifterSltToPosInUMBtmMin(p_diGoCSlt , p_diCSltToSltDist , p_diCSlt1Pos);

							ELSIF tyParamOut.diActualPosInUM > diExpectPosInUM THEN
								p_diGoCSlt		:= diExpectSlt;
								p_diMovePosInUM	:= fLifterSltToPosInUMBtmMin(p_diGoCSlt , p_diCSltToSltDist , p_diCSlt1Pos);

							ELSIF tyParamOut.diActualPosInUM < diExpectPosInUM THEN
								p_diGoCSlt		:= diExpectSlt + 1;
								p_diMovePosInUM	:= fLifterSltToPosInUMBtmMin(p_diGoCSlt , p_diCSltToSltDist , p_diCSlt1Pos);

							END_IF

							usiStep	:= 1;

						1:	//Check Position Difference
							IF tyParamOut.bPosDiff = TRUE THEN
								usiStep	:= 2;
							ELSE
								eStatus	:= Done;
							END_IF

						2:	//Move
							fbFullMovAbs.tyParamInDriver					:= tyParamInDriver;
							fbFullMovAbs.tyParamInMove.diPosInUM			:= p_diMovePosInUM;
							fbFullMovAbs.tyParamInMove.diDistInUM			:= p_diMoveDistInUM;
							fbFullMovAbs.tyParamInMove.diVelInUMPS			:= p_diMoveVelInUMPS;
							fbFullMovAbs.tyParamInMove.diAcc				:= p_diMoveAcc;
							fbFullMovAbs.tyParamInMove.diDec				:= p_diMoveDec;
							fbFullMovAbs.tyParamOut							:= tyParamOut;
							fbFullMovAbs(bEn := TRUE);

							IF fbFullMovAbs.udiStatus = 0 THEN
								eStatus	:= Done;
							ELSIF fbFullMovAbs.udiStatus < 65534 THEN
								eStatus		:= Error;

								IF fbFullMovAbs.udiStatus = 1401 THEN
									udiStatus	:= 10198;	//Power On Time Out While Going Next C Slot Position
								ELSIF fbFullMovAbs.udiStatus = 1402 THEN
									udiStatus	:= 10199;	//Homing Time Out While Going Next C Slot Position
								ELSIF fbFullMovAbs.udiStatus = 1403 THEN
									udiStatus	:= 10200;	//Move Absolute Time Out While Going Next C Slot Position
								ELSIF fbFullMovAbs.udiStatus = 1405 THEN
									udiStatus	:= 10201;	//Stop Motion Time Out While Going Next C Slot Position
								ELSIF fbFullMovAbs.udiStatus = 1408 THEN
									udiStatus	:= 10202;	//Axis Error Reset Failed While Going Next C Slot Position
								ELSIF fbFullMovAbs.udiStatus = 1409 THEN
									udiStatus	:= 10203;	//Axis Error Occur In Move Absolute While Going Next C Slot Position
								ELSIF fbFullMovAbs.udiStatus = 1411 THEN
									udiStatus	:= 10204;	//Axis Error Occur In Homing While Going Next C Slot Position
								ELSIF fbFullMovAbs.udiStatus = 1412 THEN
									udiStatus	:= 10205;	//Homing Done But Home Flag Is Not Activated While Going Next C Slot Position
								ELSIF fbFullMovAbs.udiStatus = 1413 THEN
									udiStatus	:= 10206;	//Forward Limit Activated In Homing While Going Next C Slot Position
								ELSIF fbFullMovAbs.udiStatus = 1414 THEN
									udiStatus	:= 10207;	//Reverse Limit Activated In Homing While Going Next C Slot Position
								ELSIF fbFullMovAbs.udiStatus = 1415 THEN
									udiStatus	:= 10208;	//Forward Limit Activated In Move Absolute While Going Next C Slot Position
								ELSIF fbFullMovAbs.udiStatus = 1416 THEN
									udiStatus	:= 10209;	//Reverse Limit Activated In Move Absolute While Going Next C Slot Position
								ELSE
									udiStatus	:= fbFullMovAbs.udiStatus;
								END_IF
							END_IF

					END_CASE

				END_IF

			LifterActGoPrevCSltPos:
				IF (eStatus = Idle OR eStatus = Busy) THEN

					eStatus	:= Busy;

					sStatTxt	:= a_sStatText[eStat];

					bNotInterruptible	:= TRUE;

					CASE usiStep OF
						0:	//Wait For Motion Parameter Update
							diExpectSlt		:= fLifterPosInUMToSltBtmMin(tyParamOut.diActualPosInUM , p_diCSltToSltDist , p_diCSlt1Pos);
							diExpectPosInUM	:= fLifterSltToPosInUMBtmMin(diExpectSlt , p_diCSltToSltDist , p_diCSlt1Pos);

							IF ABS(tyParamOut.diActualPosInUM - diExpectPosInUM) < 50 THEN
								p_diGoCSlt		:= diExpectSlt - 1;
								p_diMovePosInUM	:= fLifterSltToPosInUMBtmMin(p_diGoCSlt , p_diCSltToSltDist , p_diCSlt1Pos);

							ELSIF tyParamOut.diActualPosInUM > diExpectPosInUM THEN
								p_diGoCSlt		:= diExpectSlt - 1;
								p_diMovePosInUM	:= fLifterSltToPosInUMBtmMin(p_diGoCSlt , p_diCSltToSltDist , p_diCSlt1Pos);

							ELSIF tyParamOut.diActualPosInUM < diExpectPosInUM THEN
								p_diGoCSlt		:= diExpectSlt;
								p_diMovePosInUM	:= fLifterSltToPosInUMBtmMin(p_diGoCSlt , p_diCSltToSltDist , p_diCSlt1Pos);

							END_IF

							usiStep	:= 1;

						1:	//Check Position Difference
							IF tyParamOut.bPosDiff = TRUE THEN
								usiStep	:= 2;
							ELSE
								eStatus	:= Done;
							END_IF

						2:	//Move
							fbFullMovAbs.tyParamInDriver					:= tyParamInDriver;
							fbFullMovAbs.tyParamInMove.diPosInUM			:= p_diMovePosInUM;
							fbFullMovAbs.tyParamInMove.diDistInUM			:= p_diMoveDistInUM;
							fbFullMovAbs.tyParamInMove.diVelInUMPS			:= p_diMoveVelInUMPS;
							fbFullMovAbs.tyParamInMove.diAcc				:= p_diMoveAcc;
							fbFullMovAbs.tyParamInMove.diDec				:= p_diMoveDec;
							fbFullMovAbs.tyParamOut							:= tyParamOut;
							fbFullMovAbs(bEn := TRUE);

							IF fbFullMovAbs.udiStatus = 0 THEN
								eStatus	:= Done;
							ELSIF fbFullMovAbs.udiStatus < 65534 THEN
								eStatus		:= Error;

								IF fbFullMovAbs.udiStatus = 1401 THEN
									udiStatus	:= 10210;	//Power On Time Out While Going Previous C Slot Position
								ELSIF fbFullMovAbs.udiStatus = 1402 THEN
									udiStatus	:= 10211;	//Homing Time Out While Going Previous C Slot Position
								ELSIF fbFullMovAbs.udiStatus = 1403 THEN
									udiStatus	:= 10212;	//Move Absolute Time Out While Going Previous C Slot Position
								ELSIF fbFullMovAbs.udiStatus = 1405 THEN
									udiStatus	:= 10213;	//Stop Motion Time Out While Going Previous C Slot Position
								ELSIF fbFullMovAbs.udiStatus = 1408 THEN
									udiStatus	:= 10214;	//Axis Error Reset Failed While Going Previous C Slot Position
								ELSIF fbFullMovAbs.udiStatus = 1409 THEN
									udiStatus	:= 10215;	//Axis Error Occur In Move Absolute While Going Previous C Slot Position
								ELSIF fbFullMovAbs.udiStatus = 1411 THEN
									udiStatus	:= 10216;	//Axis Error Occur In Homing While Going Previous C Slot Position
								ELSIF fbFullMovAbs.udiStatus = 1412 THEN
									udiStatus	:= 10217;	//Homing Done But Home Flag Is Not Activated While Going Previous C Slot Position
								ELSIF fbFullMovAbs.udiStatus = 1413 THEN
									udiStatus	:= 10218;	//Forward Limit Activated In Homing While Going Previous C Slot Position
								ELSIF fbFullMovAbs.udiStatus = 1414 THEN
									udiStatus	:= 10219;	//Reverse Limit Activated In Homing While Going Previous C Slot Position
								ELSIF fbFullMovAbs.udiStatus = 1415 THEN
									udiStatus	:= 10220;	//Forward Limit Activated In Move Absolute While Going Previous C Slot Position
								ELSIF fbFullMovAbs.udiStatus = 1416 THEN
									udiStatus	:= 10221;	//Reverse Limit Activated In Move Absolute While Going Previous C Slot Position
								ELSE
									udiStatus	:= fbFullMovAbs.udiStatus;
								END_IF
							END_IF

					END_CASE

				END_IF

			LifterActGoDSltPos:
				IF (eStatus = Idle OR eStatus = Busy) THEN

					eStatus	:= Busy;

					sStatTxt	:= a_sStatText[eStat];

					bNotInterruptible	:= TRUE;

					CASE usiStep OF
						0:	//Wait For Motion Parameter Update
							p_diMovePosInUM	:= fLifterSltToPosInUMBtmMin(p_diGoDSlt , p_diDSltToSltDist , p_diDSlt1Pos);
							usiStep	:= 1;

						1:	//Check Position Difference
							IF tyParamOut.bPosDiff = TRUE THEN
								usiStep	:= 2;
							ELSE
								eStatus	:= Done;
							END_IF

						2:	//Move
							fbFullMovAbs.tyParamInDriver					:= tyParamInDriver;
							fbFullMovAbs.tyParamInMove.diPosInUM			:= p_diMovePosInUM;
							fbFullMovAbs.tyParamInMove.diDistInUM			:= p_diMoveDistInUM;
							fbFullMovAbs.tyParamInMove.diVelInUMPS			:= p_diMoveVelInUMPS;
							fbFullMovAbs.tyParamInMove.diAcc				:= p_diMoveAcc;
							fbFullMovAbs.tyParamInMove.diDec				:= p_diMoveDec;
							fbFullMovAbs.tyParamOut							:= tyParamOut;
							fbFullMovAbs(bEn := TRUE);

							IF fbFullMovAbs.udiStatus = 0 THEN
								eStatus	:= Done;
							ELSIF fbFullMovAbs.udiStatus < 65534 THEN
								eStatus		:= Error;

								IF fbFullMovAbs.udiStatus = 1401 THEN
									udiStatus	:= 10222;	//Power On Time Out While Going New D Slot Position
								ELSIF fbFullMovAbs.udiStatus = 1402 THEN
									udiStatus	:= 10223;	//Homing Time Out While Going New D Slot Position
								ELSIF fbFullMovAbs.udiStatus = 1403 THEN
									udiStatus	:= 10224;	//Move Absolute Time Out While Going New D Slot Position
								ELSIF fbFullMovAbs.udiStatus = 1405 THEN
									udiStatus	:= 10225;	//Stop Motion Time Out While Going New D Slot Position
								ELSIF fbFullMovAbs.udiStatus = 1408 THEN
									udiStatus	:= 10226;	//Axis Error Reset Failed While Going New D Slot Position
								ELSIF fbFullMovAbs.udiStatus = 1409 THEN
									udiStatus	:= 10227;	//Axis Error Occur In Move Absolute While Going New D Slot Position
								ELSIF fbFullMovAbs.udiStatus = 1411 THEN
									udiStatus	:= 10228;	//Axis Error Occur In Homing While Going New D Slot Position
								ELSIF fbFullMovAbs.udiStatus = 1412 THEN
									udiStatus	:= 10229;	//Homing Done But Home Flag Is Not Activated While Going New D Slot Position
								ELSIF fbFullMovAbs.udiStatus = 1413 THEN
									udiStatus	:= 10230;	//Forward Limit Activated In Homing While Going New D Slot Position
								ELSIF fbFullMovAbs.udiStatus = 1414 THEN
									udiStatus	:= 10231;	//Reverse Limit Activated In Homing While Going New D Slot Position
								ELSIF fbFullMovAbs.udiStatus = 1415 THEN
									udiStatus	:= 10232;	//Forward Limit Activated In Move Absolute While Going New D Slot Position
								ELSIF fbFullMovAbs.udiStatus = 1416 THEN
									udiStatus	:= 10233;	//Reverse Limit Activated In Move Absolute While Going New D Slot Position
								ELSE
									udiStatus	:= fbFullMovAbs.udiStatus;
								END_IF
							END_IF

					END_CASE

				END_IF

			LifterActGoNxtDSltPos:
				IF (eStatus = Idle OR eStatus = Busy) THEN

					eStatus	:= Busy;

					sStatTxt	:= a_sStatText[eStat];

					bNotInterruptible	:= TRUE;

					CASE usiStep OF
						0:	//Wait For Motion Parameter Update
							diExpectSlt		:= fLifterPosInUMToSltBtmMin(tyParamOut.diActualPosInUM , p_diDSltToSltDist , p_diDSlt1Pos);
							diExpectPosInUM	:= fLifterSltToPosInUMBtmMin(diExpectSlt , p_diDSltToSltDist , p_diDSlt1Pos);

							IF ABS(tyParamOut.diActualPosInUM - diExpectPosInUM) < 50 THEN
								p_diGoDSlt		:= diExpectSlt + 1;
								p_diMovePosInUM	:= fLifterSltToPosInUMBtmMin(p_diGoDSlt , p_diDSltToSltDist , p_diDSlt1Pos);

							ELSIF tyParamOut.diActualPosInUM > diExpectPosInUM THEN
								p_diGoDSlt		:= diExpectSlt;
								p_diMovePosInUM	:= fLifterSltToPosInUMBtmMin(p_diGoDSlt , p_diDSltToSltDist , p_diDSlt1Pos);

							ELSIF tyParamOut.diActualPosInUM < diExpectPosInUM THEN
								p_diGoDSlt		:= diExpectSlt + 1;
								p_diMovePosInUM	:= fLifterSltToPosInUMBtmMin(p_diGoDSlt , p_diDSltToSltDist , p_diDSlt1Pos);

							END_IF

							usiStep	:= 1;

						1:	//Check Position Difference
							IF tyParamOut.bPosDiff = TRUE THEN
								usiStep	:= 2;
							ELSE
								eStatus	:= Done;
							END_IF

						2:	//Move
							fbFullMovAbs.tyParamInDriver					:= tyParamInDriver;
							fbFullMovAbs.tyParamInMove.diPosInUM			:= p_diMovePosInUM;
							fbFullMovAbs.tyParamInMove.diDistInUM			:= p_diMoveDistInUM;
							fbFullMovAbs.tyParamInMove.diVelInUMPS			:= p_diMoveVelInUMPS;
							fbFullMovAbs.tyParamInMove.diAcc				:= p_diMoveAcc;
							fbFullMovAbs.tyParamInMove.diDec				:= p_diMoveDec;
							fbFullMovAbs.tyParamOut							:= tyParamOut;
							fbFullMovAbs(bEn := TRUE);

							IF fbFullMovAbs.udiStatus = 0 THEN
								eStatus	:= Done;
							ELSIF fbFullMovAbs.udiStatus < 65534 THEN
								eStatus		:= Error;

								IF fbFullMovAbs.udiStatus = 1401 THEN
									udiStatus	:= 10234;	//Power On Time Out While Going Next D Slot Position
								ELSIF fbFullMovAbs.udiStatus = 1402 THEN
									udiStatus	:= 10235;	//Homing Time Out While Going Next D Slot Position
								ELSIF fbFullMovAbs.udiStatus = 1403 THEN
									udiStatus	:= 10236;	//Move Absolute Time Out While Going Next D Slot Position
								ELSIF fbFullMovAbs.udiStatus = 1405 THEN
									udiStatus	:= 10237;	//Stop Motion Time Out While Going Next D Slot Position
								ELSIF fbFullMovAbs.udiStatus = 1408 THEN
									udiStatus	:= 10238;	//Axis Error Reset Failed While Going Next D Slot Position
								ELSIF fbFullMovAbs.udiStatus = 1409 THEN
									udiStatus	:= 10239;	//Axis Error Occur In Move Absolute While Going Next D Slot Position
								ELSIF fbFullMovAbs.udiStatus = 1411 THEN
									udiStatus	:= 10240;	//Axis Error Occur In Homing While Going Next D Slot Position
								ELSIF fbFullMovAbs.udiStatus = 1412 THEN
									udiStatus	:= 10241;	//Homing Done But Home Flag Is Not Activated While Going Next D Slot Position
								ELSIF fbFullMovAbs.udiStatus = 1413 THEN
									udiStatus	:= 10242;	//Forward Limit Activated In Homing While Going Next D Slot Position
								ELSIF fbFullMovAbs.udiStatus = 1414 THEN
									udiStatus	:= 10243;	//Reverse Limit Activated In Homing While Going Next D Slot Position
								ELSIF fbFullMovAbs.udiStatus = 1415 THEN
									udiStatus	:= 10244;	//Forward Limit Activated In Move Absolute While Going Next D Slot Position
								ELSIF fbFullMovAbs.udiStatus = 1416 THEN
									udiStatus	:= 10245;	//Reverse Limit Activated In Move Absolute While Going Next D Slot Position
								ELSE
									udiStatus	:= fbFullMovAbs.udiStatus;
								END_IF
							END_IF

					END_CASE

				END_IF

			LifterActGoPrevDSltPos:
				IF (eStatus = Idle OR eStatus = Busy) THEN

					eStatus	:= Busy;

					sStatTxt	:= a_sStatText[eStat];

					bNotInterruptible	:= TRUE;

					CASE usiStep OF
						0:	//Wait For Motion Parameter Update
							diExpectSlt		:= fLifterPosInUMToSltBtmMin(tyParamOut.diActualPosInUM , p_diDSltToSltDist , p_diDSlt1Pos);
							diExpectPosInUM	:= fLifterSltToPosInUMBtmMin(diExpectSlt , p_diDSltToSltDist , p_diDSlt1Pos);

							IF ABS(tyParamOut.diActualPosInUM - diExpectPosInUM) < 50 THEN
								p_diGoDSlt		:= diExpectSlt - 1;
								p_diMovePosInUM	:= fLifterSltToPosInUMBtmMin(p_diGoDSlt , p_diDSltToSltDist , p_diDSlt1Pos);

							ELSIF tyParamOut.diActualPosInUM > diExpectPosInUM THEN
								p_diGoDSlt		:= diExpectSlt - 1;
								p_diMovePosInUM	:= fLifterSltToPosInUMBtmMin(p_diGoDSlt , p_diDSltToSltDist , p_diDSlt1Pos);

							ELSIF tyParamOut.diActualPosInUM < diExpectPosInUM THEN
								p_diGoDSlt		:= diExpectSlt;
								p_diMovePosInUM	:= fLifterSltToPosInUMBtmMin(p_diGoDSlt , p_diDSltToSltDist , p_diDSlt1Pos);

							END_IF

							usiStep	:= 1;

						1:	//Check Position Difference
							IF tyParamOut.bPosDiff = TRUE THEN
								usiStep	:= 2;
							ELSE
								eStatus	:= Done;
							END_IF

						2:	//Move
							fbFullMovAbs.tyParamInDriver					:= tyParamInDriver;
							fbFullMovAbs.tyParamInMove.diPosInUM			:= p_diMovePosInUM;
							fbFullMovAbs.tyParamInMove.diDistInUM			:= p_diMoveDistInUM;
							fbFullMovAbs.tyParamInMove.diVelInUMPS			:= p_diMoveVelInUMPS;
							fbFullMovAbs.tyParamInMove.diAcc				:= p_diMoveAcc;
							fbFullMovAbs.tyParamInMove.diDec				:= p_diMoveDec;
							fbFullMovAbs.tyParamOut							:= tyParamOut;
							fbFullMovAbs(bEn := TRUE);

							IF fbFullMovAbs.udiStatus = 0 THEN
								eStatus	:= Done;
							ELSIF fbFullMovAbs.udiStatus < 65534 THEN
								eStatus		:= Error;

								IF fbFullMovAbs.udiStatus = 1401 THEN
									udiStatus	:= 10246;	//Power On Time Out While Going Previous D Slot Position
								ELSIF fbFullMovAbs.udiStatus = 1402 THEN
									udiStatus	:= 10247;	//Homing Time Out While Going Previous D Slot Position
								ELSIF fbFullMovAbs.udiStatus = 1403 THEN
									udiStatus	:= 10248;	//Move Absolute Time Out While Going Previous D Slot Position
								ELSIF fbFullMovAbs.udiStatus = 1405 THEN
									udiStatus	:= 10249;	//Stop Motion Time Out While Going Previous D Slot Position
								ELSIF fbFullMovAbs.udiStatus = 1408 THEN
									udiStatus	:= 10250;	//Axis Error Reset Failed While Going Previous D Slot Position
								ELSIF fbFullMovAbs.udiStatus = 1409 THEN
									udiStatus	:= 10251;	//Axis Error Occur In Move Absolute While Going Previous D Slot Position
								ELSIF fbFullMovAbs.udiStatus = 1411 THEN
									udiStatus	:= 10252;	//Axis Error Occur In Homing While Going Previous D Slot Position
								ELSIF fbFullMovAbs.udiStatus = 1412 THEN
									udiStatus	:= 10253;	//Homing Done But Home Flag Is Not Activated While Going Previous D Slot Position
								ELSIF fbFullMovAbs.udiStatus = 1413 THEN
									udiStatus	:= 10254;	//Forward Limit Activated In Homing While Going Previous D Slot Position
								ELSIF fbFullMovAbs.udiStatus = 1414 THEN
									udiStatus	:= 10255;	//Reverse Limit Activated In Homing While Going Previous D Slot Position
								ELSIF fbFullMovAbs.udiStatus = 1415 THEN
									udiStatus	:= 10256;	//Forward Limit Activated In Move Absolute While Going Previous D Slot Position
								ELSIF fbFullMovAbs.udiStatus = 1416 THEN
									udiStatus	:= 10257;	//Reverse Limit Activated In Move Absolute While Going Previous D Slot Position
								ELSE
									udiStatus	:= fbFullMovAbs.udiStatus;
								END_IF
							END_IF

					END_CASE

				END_IF

			LifterActFullHm:
				IF (eStatus = Idle OR eStatus = Busy) THEN

					eStatus	:= Busy;

					sStatTxt	:= a_sStatText[eStat];

					bNotInterruptible	:= TRUE;

					fbFullHm.tyParamInDriver	:= tyParamInDriver;
					fbFullHm.tyParamOut			:= tyParamOut;
					fbFullHm(bEn := TRUE);

					IF fbFullHm.udiStatus = 0 THEN
						eStatus	:= Done;
					ELSIF fbFullHm.udiStatus < 65534 THEN
						eStatus		:= Error;

						IF fbFullHm.udiStatus = 1401 THEN
							udiStatus	:= 10014;	//Power On Time Out While Full Homing
						ELSIF fbFullHm.udiStatus = 1402 THEN
							udiStatus	:= 10015;	//Homing Time Out While Full Homing
						ELSIF fbFullHm.udiStatus = 1405 THEN
							udiStatus	:= 10016;	//Stop Motion Time Out While Full Homing
						ELSIF fbFullHm.udiStatus = 1408 THEN
							udiStatus	:= 10017;	//Axis Error Reset Failed While Full Homing
						ELSIF fbFullHm.udiStatus = 1411 THEN
							udiStatus	:= 10018;	//Axis Error Occur In Homing While Full Homing
						ELSIF fbFullHm.udiStatus = 1412 THEN
							udiStatus	:= 10019;	//Homing Done But Home Flag Is Not Activated While Full Homing
						ELSIF fbFullHm.udiStatus = 1413 THEN
							udiStatus	:= 10020;	//Forward Limit Activated In Homing While Full Homing
						ELSIF fbFullHm.udiStatus = 1414 THEN
							udiStatus	:= 10021;	//Reverse Limit Activated In Homing While Full Homing
						ELSE
							udiStatus	:= fbFullHm.udiStatus;
						END_IF
					END_IF

				END_IF

			LifterActFullMovRel:
				IF (eStatus = Idle OR eStatus = Busy) THEN

					eStatus	:= Busy;

					sStatTxt	:= a_sStatText[eStat];

					bNotInterruptible	:= TRUE;

					fbFullMovRel.tyParamInDriver					:= tyParamInDriver;
					fbFullMovRel.tyParamInMove.diPosInUM			:= p_diMovePosInUM;
					fbFullMovRel.tyParamInMove.diDistInUM			:= p_diMoveDistInUM;
					fbFullMovRel.tyParamInMove.diVelInUMPS			:= p_diMoveVelInUMPS;
					fbFullMovRel.tyParamOut							:= tyParamOut;
					fbFullMovRel(bEn := TRUE);

					IF fbFullMovRel.udiStatus = 0 THEN
						eStatus	:= Done;
					ELSIF fbFullMovRel.udiStatus < 65534 THEN
						eStatus		:= Error;

						IF fbFullMovRel.udiStatus = 1401 THEN
							udiStatus	:= 10259;	//Power On Time Out While Full Moving Relative
						ELSIF fbFullMovRel.udiStatus = 1404 THEN
							udiStatus	:= 10260;	//Move Relative Time Out Full Moving Relative
						ELSIF fbFullMovRel.udiStatus = 1405 THEN
							udiStatus	:= 10261;	//Stop Motion Time Out While Full Moving Relative
						ELSIF fbFullMovRel.udiStatus = 1408 THEN
							udiStatus	:= 10262;	//Axis Error Reset Failed While Full Moving Relative
						ELSE
							udiStatus	:= fbFullMovRel.udiStatus;
						END_IF
					END_IF

				END_IF

			LifterActPwrOn:
				IF (eStatus = Idle OR eStatus = Busy) THEN

					eStatus	:= Busy;

					sStatTxt	:= a_sStatText[eStat];

					fbPwrOn.tyParamInDriver	:= tyParamInDriver;
					fbPwrOn(bEn := TRUE);

					IF fbPwrOn.udiStatus = 0 THEN
						eStatus	:= Done;
					ELSIF fbPwrOn.udiStatus < 65534 THEN
						eStatus		:= Error;

						IF fbPwrOn.udiStatus = 1401 THEN
							udiStatus	:= 10022;	//Power On Time Out
						ELSE
							udiStatus	:= fbPwrOn.udiStatus;
						END_IF
					END_IF

				END_IF

			LifterActPwrOff:
				IF (eStatus = Idle OR eStatus = Busy) THEN

					eStatus	:= Busy;

					sStatTxt	:= a_sStatText[eStat];

					fbPwrOff.tyParamInDriver	:= tyParamInDriver;
					fbPwrOff(bEn := TRUE);

					IF fbPwrOff.udiStatus = 0 THEN
						eStatus	:= Done;
					ELSIF fbPwrOff.udiStatus < 65534 THEN
						eStatus		:= Error;

						IF fbPwrOff.udiStatus = 1400 THEN
							udiStatus	:= 10023;	//Power Off Time Out
						ELSE
							udiStatus	:= fbPwrOff.udiStatus;
						END_IF
					END_IF

				END_IF

			LifterActHoming:
				IF (eStatus = Idle OR eStatus = Busy) THEN

					eStatus	:= Busy;

					sStatTxt	:= a_sStatText[eStat];

					bNotInterruptible	:= TRUE;

					fbHoming.tyParamInDriver	:= tyParamInDriver;
					fbHoming.tyParamOut			:= tyParamOut;
					fbHoming(bEn := TRUE);

					IF fbHoming.udiStatus = 0 THEN
						eStatus	:= Done;
					ELSIF fbHoming.udiStatus < 65534 THEN
						eStatus		:= Error;

						IF fbHoming.udiStatus = 1402 THEN
							udiStatus	:= 10024;	//Homing Time Out
						ELSIF fbHoming.udiStatus = 1411 THEN
							udiStatus	:= 10018;	//Axis Error Occur In Homing While Full Homing

						ELSIF fbHoming.udiStatus = 1413 THEN
							udiStatus	:= 10020;	//Forward Limit Activated In Homing While Full Homing
						ELSIF fbHoming.udiStatus = 1414 THEN
							udiStatus	:= 10021;	//Reverse Limit Activated In Homing While Full Homing
						ELSE
							udiStatus	:= fbHoming.udiStatus;
						END_IF
					END_IF

				END_IF

			LifterActMovAbs:
				IF (eStatus = Idle OR eStatus = Busy) THEN

					eStatus	:= Busy;

					sStatTxt	:= a_sStatText[eStat];

					bNotInterruptible	:= TRUE;

					fbMovAbs.tyParamInDriver					:= tyParamInDriver;
					fbMovAbs.tyParamInMove.diPosInUM			:= p_diMovePosInUM;
					fbMovAbs.tyParamInMove.diDistInUM			:= p_diMoveDistInUM;
					fbMovAbs.tyParamInMove.diVelInUMPS			:= p_diMoveVelInUMPS;
					fbFullMovAbs.tyParamInMove.diAcc				:= p_diMoveAcc;
					fbFullMovAbs.tyParamInMove.diDec				:= p_diMoveDec;
					fbMovAbs(bEn := TRUE);

					IF fbMovAbs.udiStatus = 0 THEN
						eStatus	:= Done;
					ELSIF fbMovAbs.udiStatus < 65534 THEN
						eStatus		:= Error;

						IF fbMovAbs.udiStatus = 1403 THEN
							udiStatus	:= 10025;	//Move Absolute Time Out
						ELSE
							udiStatus	:= fbMovAbs.udiStatus;
						END_IF
					END_IF

				END_IF

			LifterActMovRel:
				IF (eStatus = Idle OR eStatus = Busy) THEN

					eStatus	:= Busy;

					sStatTxt	:= a_sStatText[eStat];

					bNotInterruptible	:= TRUE;

					fbMovRel.tyParamInDriver					:= tyParamInDriver;
					fbMovRel.tyParamInMove.diPosInUM			:= p_diMovePosInUM;
					fbMovRel.tyParamInMove.diDistInUM			:= p_diMoveDistInUM;
					fbMovRel.tyParamInMove.diVelInUMPS			:= p_diMoveVelInUMPS;
					fbMovRel.tyParamInMove.diAcc				:= p_diMoveAcc;
					fbMovRel.tyParamInMove.diDec				:= p_diMoveDec;
					fbMovRel(bEn := TRUE);

					IF fbMovRel.udiStatus = 0 THEN
						eStatus	:= Done;
					ELSIF fbMovRel.udiStatus < 65534 THEN
						eStatus		:= Error;

						IF fbMovRel.udiStatus = 1404 THEN
							udiStatus	:= 10026;	//Move Relative Time Out
						ELSE
							udiStatus	:= fbMovRel.udiStatus;
						END_IF
					END_IF

				END_IF

			LifterActJogUp:
				IF (eStatus = Idle OR eStatus = Busy) THEN

					eStatus	:= Busy;

					sStatTxt	:= a_sStatText[eStat];

				//	bNotInterruptible	:= TRUE;

					fbJog.tyParamInDriver	:= tyParamInDriver;
					fbJog.tyParamInMove.diAcc		:= p_diMoveAcc;
					fbJog.tyParamInMove.diDec		:= p_diMoveDec;

					IF p_bDir = TRUE THEN
						fbJog.tyParamInJog.diVelInUMPS	:= p_diJogVelInUMPS * -1;
					ELSE
						fbJog.tyParamInJog.diVelInUMPS	:= p_diJogVelInUMPS;
					END_IF

					fbJog(bEn := TRUE);

					IF fbJog.udiStatus = 0 THEN
						bJogging	:= TRUE;
						eStatus		:= Done;
					ELSIF fbJog.udiStatus < 65534 THEN
						udiStatus	:= fbJog.udiStatus;
						eStatus		:= Error;
					END_IF

				END_IF

			LifterActJogDown:
				IF (eStatus = Idle OR eStatus = Busy) THEN

					eStatus	:= Busy;

					sStatTxt	:= a_sStatText[eStat];

					bNotInterruptible	:= TRUE;

					fbJog.tyParamInDriver	:= tyParamInDriver;
					fbJog.tyParamInMove.diAcc		:= p_diMoveAcc;
					fbJog.tyParamInMove.diDec		:= p_diMoveDec;

					IF p_bDir = TRUE THEN
						fbJog.tyParamInJog.diVelInUMPS	:= p_diJogVelInUMPS;
					ELSE
						fbJog.tyParamInJog.diVelInUMPS	:= p_diJogVelInUMPS * -1;
					END_IF

					fbJog(bEn := TRUE);

					IF fbJog.udiStatus = 0 THEN
						bJogging	:= TRUE;
						eStatus		:= Done;
					ELSIF fbJog.udiStatus < 65534 THEN
						udiStatus	:= fbJog.udiStatus;
						eStatus		:= Error;
					END_IF

				END_IF

			LifterActJogStop:
				IF (eStatus = Idle OR eStatus = Busy) THEN

					sStatTxt	:= a_sStatText[eStat];

					fMotionCANJogStop(ADR(tyParamOutDriver));
					bJogging	:= FALSE;

					eStatus	:= Done;

				END_IF

			LifterActRstAxisErr:
				IF (eStatus = Idle OR eStatus = Busy) THEN

					eStatus	:= Busy;

					sStatTxt	:= a_sStatText[eStat];

					fbRstAxisErr(bEn := TRUE);

					IF fbRstAxisErr.udiStatus = 0 THEN
						eStatus	:= Done;
					ELSIF fbRstAxisErr.udiStatus < 65534 THEN
						udiStatus	:= fbRstAxisErr.udiStatus;
						eStatus		:= Error;
					END_IF

				END_IF

			LifterActStop:
				IF (eStatus = Idle OR eStatus = Busy) THEN

					eStatus	:= Busy;

					sStatTxt	:= a_sStatText[eStat];

					fbStop.tyParamInDriver	:= tyParamInDriver;
					fbStop(bEn := TRUE);

					IF fbStop.udiStatus = 0 THEN
						bJogging	:= FALSE;
						eStatus		:= Done;
					ELSIF fbStop.udiStatus < 65534 THEN
						eStatus		:= Error;

						IF fbStop.udiStatus = 1405 THEN
							udiStatus	:= 10027;	//Stop Motion Time Out
						ELSE
							udiStatus	:= fbStop.udiStatus;
						END_IF
					END_IF

				END_IF
		END_CASE
ELSE
	CASE eStat OF
		LifterActSDOWrite:
			IF (eStatus = Idle OR eStatus = Busy) THEN

				eStatus	:= Busy;

				sStatTxt	:= a_sStatText[eStat];

				fbTm(IN := TRUE);

				IF fbTm.Q THEN

					fbSDOWrite.tyParamOut	:= tyParamOut;
					fbSDOWrite.tyTuning		:= p_tyTuning;
					fbSDOWrite(bEn := TRUE);

					IF fbSDOWrite.udiStatus = 0 THEN
						eStatus	:= Done;
					ELSIF fbSDOWrite.udiStatus < 65534 THEN
						fMotionCANRstCtrlWord(ADR(tyParamOutDriver));

						IF usiCount < 5 THEN
							fbTm(IN := FALSE);
							fbSDOWrite(bEn := FALSE);

							usiCount	:= usiCount + 1;
						ELSE
							eStatus		:= Error;

							IF fbSDOWrite.udiStatus = 1406 THEN
								udiStatus	:= 10028;	//SDO Write Error
							ELSE
								udiStatus	:= fbSDOWrite.udiStatus;
							END_IF
						END_IF

					END_IF

				END_IF

			END_IF

		LifterActBGStartModOKChk:
			IF (eStatus = Idle OR eStatus = Busy) THEN

				sStatTxt	:= a_sStatText[eStat];

				bModuleOKChk	:= TRUE;
				eStatus			:= Done;

			END_IF

		LifterActBGStopModOKChk:
			IF (eStatus = Idle OR eStatus = Busy) THEN

				sStatTxt	:= a_sStatText[eStat];

				bModuleOKChk	:= FALSE;
				eStatus			:= Done;

			END_IF

		LifterActIdle:
			IF eStatus <> Idle THEN	//Reset Data
				//Private
				fbStop(bEn := FALSE);
				fbRstAxisErr(bEn := FALSE);
				fbJog(bEn := FALSE);
				fbMovRel(bEn := FALSE);
				fbMovAbs(bEn := FALSE);
				fbHoming(bEn := FALSE);
				fbPwrOff(bEn := FALSE);
				fbPwrOn(bEn := FALSE);
				fbFullHm(bEn := FALSE);
				fbFullMovAbs(bEn := FALSE);
				fbSDOWrite(bEn := FALSE);
				fbTm(IN := FALSE);
				usiStep				:= 0;
				usiCount			:= 0;
				bNotInterruptible	:= FALSE;

				sStatTxt	:= a_sStatText[eStat];

			END_IF

			eStatus	:= Idle;

			IF EDGENEG(p_bManual) THEN
				fMotionCANRstCtrlWord(ADR(tyParamOutDriver));
			END_IF

		LifterActRstNode:
			IF (eStatus = Idle OR eStatus = Busy) THEN

				eStatus	:= Busy;

				sStatTxt	:= a_sStatText[eStat];
				IF bRstErr THEN
					fbModuleOK(bEn := FALSE, bModuleOK := bModuleOK);
				END_IF
				fbModuleOK(bEn := TRUE);
				IF fbModuleOK.udiStatus = 0 THEN
					fbModuleOK(bEn := FALSE);
					eStatus			:= Done;
				ELSIF fbModuleOK.udiStatus < 65534 THEN
					eStatus		:= Error;

					IF fbModuleOK.udiStatus = 1407 THEN
						udiStatus	:= 10001;	//CANOpen Communication Error, ModuleOK Not TRUE
						fbModuleOK(bEn := FALSE);
					ELSE
						udiStatus	:= fbModuleOK.udiStatus;
					END_IF
				END_IF
			END_IF

		LifterActRstAxisErr:
			IF (eStatus = Idle OR eStatus = Busy) THEN

				eStatus	:= Busy;

				sStatTxt	:= a_sStatText[eStat];

				fbRstAxisErr(bEn := TRUE);

				IF fbRstAxisErr.udiStatus = 0 THEN
					eStatus	:= Done;
				ELSIF fbRstAxisErr.udiStatus < 65534 THEN
					udiStatus	:= fbRstAxisErr.udiStatus;
					eStatus		:= Error;
				END_IF

			END_IF

		END_CASE

	END_IF

	//added
	iLifterMovedSlot := BOOL_TO_USINT(eStat = LifterActGoASltPos)*1+
						BOOL_TO_USINT(eStat = LifterActGoBSltPos)*2+
						BOOL_TO_USINT(eStat = LifterActGoCSltPos)*3;

END_ACTION
```

#### Act_Main_Disable.st - Do Not Change!!!
```iecst
(** 2020-03-16 **)
ACTION Act_Main_Disable:

	tyParamOut.bAxisErr			:= FALSE;
	tyParamOut.bFwdLmtSen		:= FALSE;
	tyParamOut.bInPos			:= TRUE;
	tyParamOut.bIsHomed			:= TRUE;
	tyParamOut.bPosDiff			:= FALSE;
	tyParamOut.bPwrOn			:= TRUE;
	tyParamOut.bRevLmtSen		:= FALSE;
	tyParamOut.bStopped			:= TRUE;
	tyParamOut.diActualPosInUM	:= 0;
	tyParamOut.diHmAcc			:= 0;
	tyParamOut.diHmSpdForSwitch	:= 0;
	tyParamOut.diHmSpdForZero	:= 0;
	tyParamOut.diProfileAcc		:= 0;
	tyParamOut.diProfileDec		:= 0;
	tyParamOut.udiAxisErrID		:= 0;

	bSltAPosDiff				:= FALSE;
	bSltBPosDiff				:= FALSE;
	bSltCPosDiff				:= FALSE;
	bSltDPosDiff				:= FALSE;
	bModuleNotOK				:= FALSE;
END_ACTION
```

#### Act_Background.st - Do Not Change!!!
```iecst
(** 2020-03-20 **)
ACTION Act_Background:

	//Update Parameter
	IF bModuleOK = TRUE THEN

		tyParamInMove.diPosInUM				:= p_diMovePosInUM;
		tyParamInMove.diDistInUM			:= p_diMoveDistInUM;
		tyParamInMove.diVelInUMPS			:= p_diMoveVelInUMPS;
		tyParamInMove.diAcc			:= p_diMoveAcc;
		tyParamInMove.diDec			:= p_diMoveDec;

		fMotionCANUpdtDat(ADR(tyParamOut) , p_tyParamInConvert , tyParamOutDriver , tyParamInDriver , tyParamInMove , p_tyParamInHm , p_bDir, p_eNtParamMotorType);

		bSltAPosDiff	:= (tyParamOut.bIsHomed = FALSE) OR ((ABS((fLifterSltToPosInUMBtmMin(p_diGoASlt , p_diASltToSltDist , p_diASlt1Pos)) - tyParamOut.diActualPosInUM)) > 500);
		bSltBPosDiff	:= (tyParamOut.bIsHomed = FALSE) OR ((ABS((fLifterSltToPosInUMBtmMin(p_diGoBSlt , p_diBSltToSltDist , p_diBSlt1Pos)) - tyParamOut.diActualPosInUM)) > 500);
		bSltCPosDiff	:= (tyParamOut.bIsHomed = FALSE) OR ((ABS((fLifterSltToPosInUMBtmMin(p_diGoCSlt , p_diCSltToSltDist , p_diCSlt1Pos)) - tyParamOut.diActualPosInUM)) > 500);
		bSltDPosDiff	:= (tyParamOut.bIsHomed = FALSE) OR ((ABS((fLifterSltToPosInUMBtmMin(p_diGoDSlt , p_diDSltToSltDist , p_diDSlt1Pos)) - tyParamOut.diActualPosInUM)) > 500);
		diCurrSltA		:= fLifterPosInUMToSltBtmMin(tyParamOut.diActualPosInUM , p_diASltToSltDist , p_diASlt1Pos);
		diCurrSltB		:= fLifterPosInUMToSltBtmMin(tyParamOut.diActualPosInUM , p_diBSltToSltDist , p_diBSlt1Pos);
		diCurrSltC		:= fLifterPosInUMToSltBtmMin(tyParamOut.diActualPosInUM , p_diCSltToSltDist , p_diCSlt1Pos);
		diCurrSltD		:= fLifterPosInUMToSltBtmMin(tyParamOut.diActualPosInUM , p_diDSltToSltDist , p_diDSlt1Pos);
		bAPosDiff		:= (tyParamOut.bIsHomed = FALSE) OR ((ABS(p_diAPos - tyParamOut.diActualPosInUM)) > 500);
		bBPosDiff		:= (tyParamOut.bIsHomed = FALSE) OR ((ABS(p_diBPos - tyParamOut.diActualPosInUM)) > 500);
		bCPosDiff		:= (tyParamOut.bIsHomed = FALSE) OR ((ABS(p_diCPos - tyParamOut.diActualPosInUM)) > 500);
		bDPosDiff		:= (tyParamOut.bIsHomed = FALSE) OR ((ABS(p_diDPos - tyParamOut.diActualPosInUM)) > 500);
		bEPosDiff		:= (tyParamOut.bIsHomed = FALSE) OR ((ABS(p_diEPos - tyParamOut.diActualPosInUM)) > 500);
		bFPosDiff		:= (tyParamOut.bIsHomed = FALSE) OR ((ABS(p_diFPos - tyParamOut.diActualPosInUM)) > 500);
		bGPosDiff		:= (tyParamOut.bIsHomed = FALSE) OR ((ABS(p_diGPos - tyParamOut.diActualPosInUM)) > 500);
		bHPosDiff		:= (tyParamOut.bIsHomed = FALSE) OR ((ABS(p_diHPos - tyParamOut.diActualPosInUM)) > 500);

		IF p_bDir = TRUE THEN
			bUpSen		:= tyParamOut.bRevLmtSen;
			bDownSen	:= tyParamOut.bFwdLmtSen;
		ELSE
			bUpSen		:= tyParamOut.bFwdLmtSen;
			bDownSen	:= tyParamOut.bRevLmtSen;
		END_IF

		CASE p_eNtParamMotorType OF
			DeltaAsdaA2:
				CASE tyParamOut.udiAxisErrID OF
					8976:	sAxisErrTxt	:= 'Over Current';
					12560:	sAxisErrTxt	:= 'Over Voltage';
					12576:	sAxisErrTxt	:= 'Under Voltage';
					12592:	sAxisErrTxt	:= 'Input Power Phase Loss';
					12816:	sAxisErrTxt	:= 'Regeneration Error';
					12848:	sAxisErrTxt	:= 'Overload';
					12849:	sAxisErrTxt	:= 'Pre-overload Warning';
					13056:	sAxisErrTxt	:= 'U,V,W Wiring Error';
					16912:	sAxisErrTxt	:= 'IGBT Temperature Error';
					21296:	sAxisErrTxt	:= 'Memory Error';
					21569:	sAxisErrTxt	:= 'Emergency Stop Activated';
					21570:	sAxisErrTxt	:= 'Forward Limit Switch Error';
					21571:	sAxisErrTxt	:= 'Reverse Limit Switch Error';
					21572:	sAxisErrTxt	:= 'Forward Software Limit';
					21573:	sAxisErrTxt	:= 'Reverse Software Limit';
					21760:	sAxisErrTxt	:= 'DSP Firmware Upgrade';
					25088:	sAxisErrTxt	:= 'CANopen SYNC Error';
					25360:	sAxisErrTxt	:= 'CANopen Data Initial Error';
					25376:	sAxisErrTxt	:= 'Adjustment Error';
					28961:	sAxisErrTxt	:= 'Motor Protection Error';
					28962:	sAxisErrTxt	:= 'Motor Error';
					29445:	sAxisErrTxt	:= 'Encoder Error';
					29446:	sAxisErrTxt	:= 'Encoder Output Error';
					29968:	sAxisErrTxt	:= 'Serial Communication Error';
					29984:	sAxisErrTxt	:= 'Serial Communication Time Out';
					33024:	sAxisErrTxt	:= 'CANbus Error (Bus-off)';
					33040:	sAxisErrTxt	:= 'CANopen SDO receive buffer overrun';
					33056:	sAxisErrTxt	:= 'CANbus Error (Warning)';
					33072:	sAxisErrTxt	:= 'Node Guarding or Heartbeat Error';
					33280:	sAxisErrTxt	:= 'CANopen PDO Object Error';
					33792:	sAxisErrTxt	:= 'Over Speed';
					34304:	sAxisErrTxt	:= 'Abnormal Pulse Control Command';
					34320:	sAxisErrTxt	:= 'Full Closed Loop Excessive Deviation';
					34321:	sAxisErrTxt	:= 'Excessive Deviation';
				END_CASE

			SchneiderLexium28:
				CASE tyParamOut.udiAxisErrID OF
					8724:	sAxisErrTxt	:= 'Over Current';
					8976:	sAxisErrTxt	:= 'Motor Overload';
					8977:	sAxisErrTxt	:= 'Drive overload (foldback)';
					9088:	sAxisErrTxt	:= 'Calculated offsets for current sensors out OF range';
					9089:	sAxisErrTxt := 'Motor phase missing';
					9090:	sAxisErrTxt := 'Overcurrent detected at one OF the digital outputs';
					12560:	sAxisErrTxt	:= 'DC Bus Over Voltage';
					12576:	sAxisErrTxt	:= 'DC Bus Under Voltage';
					12672:	sAxisErrTxt	:= 'Braking Resistor Overload';
					12673:	sAxisErrTxt	:= 'Safety function Safe Torque Off (STO) triggered';
					12674:	sAxisErrTxt	:= 'DC bus voltage measurement';
					12675:	sAxisErrTxt	:= 'Missing mains supply, undervoltage mains supply';
					12676:	sAxisErrTxt := 'The encoder supply voltage has dropped under operational value';
					12677:	sAxisErrTxt := 'The multi turn encoder battery voltage has dropped under 3 Vdc';
					12678:	sAxisErrTxt := 'Internal position synchronization error	detected between the multi turn AND the single turn modules';
					12679:	sAxisErrTxt := 'Generic error code of the multi turn module is detected';
					12697:	sAxisErrTxt := 'Braking resistor overload';
					16512:	sAxisErrTxt	:= 'Drive overtemperature (IPM)';
					16513:	sAxisErrTxt	:= 'Drive overtemperature (controller)';
					16534:	sAxisErrTxt := 'Temperature sensor inoperative';
					17168:	sAxisErrTxt	:= 'Power stage overtemperature';
					17280:	sAxisErrTxt := 'The encoder temperature is too high';
					17424:	sAxisErrTxt	:= 'Motor overtemperature';
					21808:	sAxisErrTxt	:= 'System error detected (nonvolatilememory)';
					21893:	sAxisErrTxt	:= 'Error detected in non-volatile memory';
					21889:	sAxisErrTxt	:= 'System error detected (nonvolatile memory)';
					21890:	sAxisErrTxt	:= 'System error detected (CAN power supply)';
					21891:	sAxisErrTxt	:= 'System error detected (selftest)';
					21894:	sAxisErrTxt	:= 'System error detected (NV ACCESS)';
					25472:	sAxisErrTxt	:= 'Target position rejected';
					25985:	sAxisErrTxt	:= 'System error detected(FPGA)';
					28816:	sAxisErrTxt	:= 'System error detected (FPGA does NOT match firmware)';
					28817:	sAxisErrTxt	:= 'Emergency Stop Activated';
					28961:	sAxisErrTxt := 'Motor blocked';
					29080:	sAxisErrTxt := 'Commutation error detected';
					29568:  sAxisErrTxt	:= 'Error detected in communication with motor encoder';
					29574:	sAxisErrTxt	:= 'Drive is not synchronous wit master cycle';
					29581:	sAxisErrTxt := 'System error detected (encoder)';
					29587:	sAxisErrTxt	:= 'Encoder overvoltage or overcurrent';
					29592:	sAxisErrTxt := 'The returned position value are no longer considered valid';
					29593:	sAxisErrTxt := 'The multi turn encoder requires an explicit configuration command';
					30081:	sAxisErrTxt := 'Target position rejected';
					30082:	sAxisErrTxt := 'No target values received via the fieldbus';
					33072:	sAxisErrTxt	:= 'CANopen: Heartbeat error detected';
					33296:	sAxisErrTxt := 'R_PDO is too short';
					33921:	sAxisErrTxt	:= 'Actual Motor Velocity Too High';
					33553:	sAxisErrTxt	:= 'Motor torque too high FOR an excessive period OF time';
					33664:	sAxisErrTxt := 'Unstable current loop';
					33922:	sAxisErrTxt := 'Velocity deviation too high';
					34321:	sAxisErrTxt	:= 'Position deviation too high';
					34432:	sAxisErrTxt := 'Position deviation via signal output function MC_OK';
					34441:	sAxisErrTxt := 'Position deviation too high (following error)';
					61568:	sAxisErrTxt	:= 'Fieldbus: Communication	error detected';
					65282:	sAxisErrTxt	:= 'Not possible to read data of electronic motor nameplate';
					65296:	sAxisErrTxt	:= 'Forward Limit Switch Error';
					65297:	sAxisErrTxt	:= 'Reverse Limit Switch Error';
					65281:	sAxisErrTxt := 'System error detected';
					65298:	sAxisErrTxt	:= 'Forward Software Limit';
					65299:	sAxisErrTxt	:= 'Reverse Software Limit';
					65301:	sAxisErrTxt := 'The encoder firmware cannot operate on the provided hardware';

				END_CASE

			EstunPronet:
				CASE tyParamOut.udiAxisErrID OF
					65281:	sAxisErrTxt	:= 'Parameter breakdown';//A01
					65282:	sAxisErrTxt	:= 'AD shift channels breakdown';
					65283:	sAxisErrTxt	:= 'Overspeed';
					65284:	sAxisErrTxt	:= 'Overload';
					65285:	sAxisErrTxt := 'Position error counteroverflow ';
					65286:	sAxisErrTxt := 'Position error pulse overflow';
					65287:	sAxisErrTxt	:= 'The setting of electronic gear or given pulse frequency is not reasonable';
					65288:	sAxisErrTxt	:= 'The 1st channel of current detection is wrong.';
					65289:	sAxisErrTxt	:= 'The 2nd channel of current detection is wrong.';
					65290:	sAxisErrTxt	:= 'Incremental Encoder is break off.';//A10
					65292:	sAxisErrTxt	:= 'Overcurrent';
					65293:	sAxisErrTxt	:= 'Overvoltage';
					65294:	sAxisErrTxt	:= 'Undervoltage';
					65295:	sAxisErrTxt := 'Bleeder resistor error';
					65296:	sAxisErrTxt := 'Regeneration error';
					65297:	sAxisErrTxt := 'Resolver error';
					65298:	sAxisErrTxt := 'IGBT superheat alarm';
					65299:	sAxisErrTxt := 'Motor overheat alarm';
					65300:	sAxisErrTxt := 'Power line phase shortage';//A20
					65301:	sAxisErrTxt	:= 'Instantaneous power off alarm';
					65302:	sAxisErrTxt	:= 'Motor temperature detection sensor is break off.';
					65303:	sAxisErrTxt := 'Brake overcurrent alarm';//A23
					65305:	sAxisErrTxt := 'Motor power line U overcurrent';//A25
					65306:	sAxisErrTxt := 'Motor power line V overcurrent';//A26
					65307:	sAxisErrTxt := 'Motor power line W overcurrent';//A27
					65322:	sAxisErrTxt	:= 'Servomotor type error';//A42
					65323:	sAxisErrTxt	:= 'Servo drive type error';
					65325:	sAxisErrTxt	:= 'Absolute encoder multiturn information error';
					65326:	sAxisErrTxt	:= 'Absolute encoder multiturn information overflow';
					65327:	sAxisErrTxt	:= 'Battery voltage below 2.5V';
					65328:	sAxisErrTxt	:= 'Battery voltage below 3.1V';//A48
					65330:	sAxisErrTxt := 'Serial encoder communication overtime ';//A50
					65331:	sAxisErrTxt := 'Absolute encoder overspeed alarm detected';
					65332:  sAxisErrTxt	:= 'Absolute state of serial encoder error';
					65333:	sAxisErrTxt	:= 'Serial encoder calcaution error';
					65334:	sAxisErrTxt := 'Parity bit or end bit in serial encoder control domain error';
					65335:	sAxisErrTxt	:= 'Serial encoder communication data checking error';
					65336:	sAxisErrTxt := 'End bit in serial encoder control domain error';
					65338:	sAxisErrTxt := 'Serial encoder data empty';
					65339:	sAxisErrTxt := 'Serial encoder data format error';
					65340:	sAxisErrTxt := 'Communication module not detected ';//A60
					65341:	sAxisErrTxt := 'Communication unsuccessful';
					65342:	sAxisErrTxt := 'Servo drive can not receive the period data of communication module ';
					65343:	sAxisErrTxt := 'Communication module can not receive the servo drive response data.';
					65344:	sAxisErrTxt := 'Communication module and bus connectionless';
					65346:	sAxisErrTxt := 'CAN communication abnormal';
					65347:	sAxisErrTxt := 'Receiving heartbeat timeout';
					65349:	sAxisErrTxt := 'Synchronization signal monitoring cycle is longer than setting';
					65362:  sAxisErrTxt	:= 'Torque output alarm';
				END_CASE
		END_CASE
	ELSE

		tyParamOut.bAxisErr			:= FALSE;
		tyParamOut.bFwdLmtSen		:= FALSE;
		tyParamOut.bInPos			:= FALSE;
		tyParamOut.bIsHomed			:= FALSE;
		tyParamOut.bPosDiff			:= TRUE;
		tyParamOut.bPwrOn			:= FALSE;
		tyParamOut.bRevLmtSen		:= FALSE;
		tyParamOut.bStopped			:= TRUE;
		tyParamOut.diActualPosInUM	:= 0;
		tyParamOut.diHmAcc			:= 0;
		tyParamOut.diHmSpdForSwitch	:= 0;
		tyParamOut.diHmSpdForZero	:= 0;
		tyParamOut.diProfileAcc		:= 0;
		tyParamOut.diProfileDec		:= 0;
		tyParamOut.udiAxisErrID		:= 0;

		bSltAPosDiff				:= TRUE;
		bSltBPosDiff				:= TRUE;
		bSltCPosDiff				:= TRUE;
		bSltDPosDiff				:= TRUE;
		diCurrSltA					:= 0;
		diCurrSltB					:= 0;
		diCurrSltC					:= 0;
		diCurrSltD					:= 0;
		bAPosDiff					:= TRUE;
		bBPosDiff					:= TRUE;
		bCPosDiff					:= TRUE;
		bDPosDiff					:= TRUE;
		bEPosDiff					:= TRUE;
		bFPosDiff					:= TRUE;
		bGPosDiff					:= TRUE;
		bHPosDiff					:= TRUE;

	END_IF

	//Abnormal Movement
	IF eStatus1 <> Error THEN
		IF p_bOps = TRUE AND eStatus = Idle THEN
			IF (ABS(tyParamOut.diActualPosInUM - diActualPosInUMOld) > 2000) AND (ABS(tyParamOut.diActualPosInUM - diActualPosInUMOld) < 30000) THEN
				eStatus1	:= Error;
				udiStatus1	:= 10000;	//Axis Move Abnormally By External Force

				fMotionCANRstCtrlWord(ADR(tyParamOutDriver));
				p_eAct	:= LifterActIdle;
				eStat	:= LifterActIdle;
			END_IF
		ELSE
			diActualPosInUMOld	:= tyParamOut.diActualPosInUM;
		END_IF
	END_IF

	//Reset Error
	IF (eStatus1 = Error) AND bRstErr THEN
		eStatus1	:= Idle;
		udiStatus1	:= 0;
	END_IF

	//Request Position To Movement Out Of Range
	IF p_bOps
		AND((tyParamInMove.diPosInUM < p_diMinAbsPosInUM) OR (tyParamInMove.diPosInUM > p_diMaxAbsPosInUM))
		AND (eStatus2 <> Error) THEN
		eStatus2	:= Error;
		udiStatus2	:= 10077;	//Request Absolute Position Out Of Range

		fMotionCANRstCtrlWord(ADR(tyParamOutDriver));
		p_eAct	:= LifterActIdle;
		eStat	:= LifterActIdle;
	END_IF

	//Reset Error
	IF (eStatus2 = Error) AND bRstErr THEN
		eStatus2	:= Idle;
		udiStatus2	:= 0;
	END_IF

	//Sensor Interrupt
	IF bNotInterruptible = TRUE AND eStatus3 <> Error THEN

		IF p_bInterruptSensor1 OR p_bInterruptSensor2 OR p_bInterruptSensor3 OR p_bInterruptSensor4 OR p_bInterruptSensor5 OR p_bInterruptSensor6 THEN

			eStatus3	:= Error;
			udiStatus3	:= 10258;	//Sensor Interrupt Lifter Movement

			fMotionCANRstCtrlWord(ADR(tyParamOutDriver));
			p_eAct	:= LifterActIdle;
			eStat	:= LifterActIdle;
		END_IF

	END_IF

	//Reset Error
	IF (eStatus3 = Error) AND bRstErr THEN
		eStatus3	:= Idle;
		udiStatus3	:= 0;
	END_IF

	IF bRstErr THEN
		udiStatus	:= 0;
	END_IF

	fbServoModuleOk(IN:= bModuleOK);
	fbServoModuleNotOk(IN:= bModuleOK = FALSE);
	IF fbServoModuleNotOk.Q AND udiStatus <> 10001 THEN

		bModuleNotOK		:= TRUE;
		bModuleNotOKLock	:= TRUE;
		usiRstStep	:= 0;
		tyParamOutDriver.uiCtrlword_6040	:= 0;
		tyParamOutDriver.siModOfOpt_6060	:= 0;
		tyParamOutDriver.diTargetPos_607A	:= 0;
		tyParamOutDriver.udiMoveSpd_6081	:= 0;
		tyParamOutDriver.siHmMethod_6098	:= 0;
		tyParamOutDriver.diJogVel_60FF		:= 0;

		CASE p_eNtParamMotorType OF

			DeltaAsdaA2:
				fbModuleOK(bModuleOK:= FALSE);
				IF eStatus = Idle THEN
					eAct	:= LifterActRstNode;
				END_IF

				IF (eStatus = Done OR eStatus = Error)AND eStat = LifterActRstNode THEN

					eAct	:= LifterActIdle;
				END_IF

			EstunPronet:
				fbModuleOK(bModuleOK:= FALSE);
				IF eStatus = Idle THEN
					eAct	:= LifterActRstNode;
				END_IF

				IF (eStatus = Done OR eStatus = Error)AND eStat = LifterActRstNode THEN

					eAct	:= LifterActIdle;
				END_IF

			SchneiderLexium28:
			// Do Nothing
		END_CASE

	ELSIF bModuleNotOK = TRUE AND fbServoModuleOk.Q THEN

		CASE usiRstStep OF

			0:
				IF eStatus = Idle THEN
					eAct	:= LifterActRstAxisErr;
				END_IF

				IF eStatus = Done AND eStat = LifterActRstAxisErr THEN
					eAct	:= LifterActIdle;
					usiRstStep	:= 4;
				END_IF

			4: tyParamOutDriver.siModOfOpt_6060 := 1;
				usiRstStep	:= 5;

			5: tyParamOutDriver.siModOfOpt_6060 := 1;
				fbRstNodeTimer(IN:=TRUE);

				IF tyParamInDriver.siModOfOptDisp_6061 = 1 THEN
					usiRstStep	:= 6;
					fbRstNodeTimer(IN:=FALSE);
				ELSIF fbRstNodeTimer.Q THEN
					usiRstStep	:= 8;
					fbRstNodeTimer(IN:=FALSE);
				END_IF

			6: tyParamOutDriver.siModOfOpt_6060 := 6;
				fbRstNodeTimer(IN:=FALSE);
				usiRstStep	:= 7;

			7: tyParamOutDriver.siModOfOpt_6060 := 6;
				fbRstNodeTimer(IN:=TRUE);

				IF tyParamInDriver.siModOfOptDisp_6061 = 6 THEN
					usiRstStep	:= 10;
					fbRstNodeTimer(IN:=FALSE);
				ELSIF fbRstNodeTimer.Q THEN
					usiRstStep	:= 9;
					fbRstNodeTimer(IN:=FALSE);
				END_IF

			8:	fbModuleOK(bEn := TRUE, bModuleOK:= FALSE);
				fbRstNodeTimer(IN:=FALSE);
				usiRstStep	:= 9;

			9:	fbModuleOK(bModuleOK:= FALSE);
				IF eStatus = Idle THEN
					eAct	:=LifterActRstNode;
				END_IF

				IF eStatus = Done AND eStat = LifterActRstNode THEN
					usiRstStep	:= 0;
					eAct		:= LifterActIdle;
				END_IF

			10:IF eStatus = Idle THEN
					eAct	:= LifterActRstAxisErr;
				END_IF

				IF eStatus = Done AND eStat = LifterActRstAxisErr THEN
					eAct			:= LifterActIdle;
					usiRstStep	:= 11;
				END_IF

			11:

				IF eStatus = Idle THEN
					eAct	:= LifterActSDOWrite;
				END_IF

				IF eStatus = Done AND eStat = LifterActSDOWrite THEN
					eAct			:= LifterActIdle;
					usiRstStep	:= 13;

				ELSIF udiStatus = 10028 THEN
					eAct			:= LifterActIdle;
					usiRstStep	:= 0;
				END_IF

			13: bModuleNotOK	:= FALSE;
				usiRstStep	:= 0;
		END_CASE
	ELSE
		eAct	:= LifterActIdle;

	END_IF

	IF tyParamOut.bPosDiff = FALSE THEN
		tyParamOutDriver.uiCtrlword_6040.4	:= FALSE;
	END_IF

END_ACTION
```
